  MoveC 574 to (267.87, -55.04, -8.35) mm, rotated rx -180 ry 0 rz 0 deg; joints [19.614, -51.076, 148.071, 19.71, -95.718, 2.626] to (268.06, -55.49, -8.35) mm, rotated rx -180 ry 0 rz 0 deg; joints [19.592, -51.078, 148.094, 19.688, -95.739, 2.631]
  MoveL 575 to (268.06, -80.89, -8.35) mm, rotated rx -180 ry 0 rz 0 deg; joints [18.101, -51.105, 148.664, 18.209, -96.314, 2.629]
  MoveL 576 to (217.26, -80.89, -8.35) mm, rotated rx -180 ry 0 rz 0 deg; joints [17.167, -50.698, 145.241, 17.193, -93.471, 1.614]
  MoveL 577 to (217.26, -30.09, -8.35) mm, rotated rx 180 ry 0 rz 0 deg; joints [19.994, -50.561, 144.093, 20.006, -92.45, 1.48]
  MoveL 578 to (268.06, -30.09, -8.35) mm, rotated rx 180 ry 0 rz 0 deg; joints [21.056, -51.039, 147.478, 21.138, -95.138, 2.59]
  MoveL 579 to (268.06, -55.49, -8.35) mm, rotated rx -180 ry 0 rz 0 deg; joints [19.592, -51.078, 148.094, 19.688, -95.739, 2.631]
  MoveC 580 to (267.87, -55.94, -8.35) mm, rotated rx 180 ry 0 rz 0 deg; joints [19.562, -51.077, 148.092, 19.658, -95.739, 2.627] to (267.42, -56.12, -8.35) mm, rotated rx -180 ry 0 rz 0 deg; joints [19.542, -51.074, 148.066, 19.637, -95.719, 2.617]
  MoveL 581 to (266.79, -56.12, -8.35) mm, rotated rx 180 ry 0 rz 0 deg; joints [19.529, -51.07, 148.024, 19.623, -95.684, 2.603]
  MoveC 582 to (266.34, -56.12, -8.16) mm, rotated rx -180 ry 0 rz 0 deg; joints [19.519, -51.086, 147.998, 19.612, -95.645, 2.588] to (266.15, -56.12, -7.72) mm, rotated rx -180 ry 0 rz 0 deg; joints [19.515, -51.13, 147.995, 19.606, -95.6, 2.571]
  Set speed (500.0 mm/s)
  MoveL 583 to (266.15, -56.12, 6) mm, rotated rx 180 ry 0 rz 0 deg; joints [19.507, -52.51, 148.253, 19.565, -94.544, 2.193]
  MoveL 584 to (139.15, -54.85, 6) mm, rotated rx 180 ry 0 rz 0 deg; joints [17.26, -50.798, 139.522, 17.265, -87.911, -0.107]
  Set speed (25.4 mm/s)
  MoveL 585 to (139.15, -54.85, -3.54) mm, rotated rx -180 ry 0 rz 0 deg; joints [17.264, -49.983, 139.368, 17.264, -88.543, 0.09]
  MoveC 586 to (139.34, -54.85, -3.99) mm, rotated rx 180 ry 0 rz 0 deg; joints [17.268, -49.948, 139.374, 17.267, -88.582, 0.102] to (139.79, -54.85, -4.17) mm, rotated rx -180 ry 0 rz 0 deg; joints [17.275, -49.94, 139.402, 17.274, -88.617, 0.113]
  Set speed (50.8 mm/s)
  MoveL 587 to (140.42, -54.85, -4.18) mm, rotated rx 180 ry 0 rz 0 deg; joints [17.285, -49.95, 139.447, 17.284, -88.65, 0.123]
  MoveC 588 to (140.87, -55.04, -4.18) mm, rotated rx -180 ry 0 rz 0 deg; joints [17.283, -49.958, 139.482, 17.281, -88.676, 0.131] to (141.06, -55.49, -4.17) mm, rotated rx -180 ry 0 rz 0 deg; joints [17.262, -49.963, 139.505, 17.261, -88.693, 0.136]
  MoveL 589 to (141.06, -80.89, -4.17) mm, rotated rx 180 ry 0 rz 0 deg; joints [15.927, -50.066, 140.034, 15.923, -89.099, 0.263]
  MoveL 590 to (90.26, -80.89, -4.18) mm, rotated rx -180 ry 0 rz 0 deg; joints [15.195, -49.17, 136.413, 15.218, -86.47, -0.451]
  MoveL 591 to (90.26, -30.09, -4.18) mm, rotated rx -180 ry 0 rz 0 deg; joints [17.739, -48.917, 135.342, 17.784, -85.727, -0.819]
  MoveL 592 to (141.06, -30.09, -4.17) mm, rotated rx -180 ry 0 rz 0 deg; joints [18.578, -49.847, 138.934, 18.581, -88.265, -0.019]
  MoveL 593 to (141.06, -55.49, -4.18) mm, rotated rx -180 ry 0 rz 0 deg; joints [17.262, -49.963, 139.505, 17.261, -88.693, 0.136]
  MoveC 594 to (140.87, -55.94, -4.18) mm, rotated rx 180 ry 0 rz 0 deg; joints [17.236, -49.962, 139.502, 17.234, -88.691, 0.136] to (140.42, -56.12, -4.17) mm, rotated rx -180 ry 0 rz 0 deg; joints [17.219, -49.956, 139.474, 17.218, -88.671, 0.13]
  MoveL 595 to (139.79, -56.12, -4.18) mm, rotated rx 180 ry 0 rz 0 deg; joints [17.209, -49.945, 139.43, 17.208, -88.638, 0.12]
  MoveC 596 to (139.34, -56.12, -3.99) mm, rotated rx -180 ry 0 rz 0 deg; joints [17.201, -49.954, 139.401, 17.2, -88.603, 0.109] to (139.15, -56.12, -3.54) mm, rotated rx -180 ry 0 rz 0 deg; joints [17.198, -49.989, 139.396, 17.198, -88.564, 0.097]
  Set speed (500.0 mm/s)
  MoveL 597 to (139.15, -56.12, 5) mm, rotated rx -180 ry 0 rz 0 deg; joints [17.194, -50.719, 139.534, 17.199, -87.998, -0.078]
  MoveL 598 to (139.15, -54.85, 5) mm, rotated rx -180 ry 0 rz 0 deg; joints [17.26, -50.713, 139.506, 17.265, -87.978, -0.086]
  Set speed (25.4 mm/s)
  MoveL 599 to (139.15, -54.85, 1.82) mm, rotated rx -180 ry 0 rz 0 deg; joints [17.262, -50.442, 139.456, 17.264, -88.189, -0.02]
  MoveL 600 to (139.15, -54.85, -7.72) mm, rotated rx -180 ry 0 rz 0 deg; joints [17.266, -49.627, 139.298, 17.264, -88.817, 0.175]
  MoveC 601 to (139.34, -54.85, -8.16) mm, rotated rx 180 ry 0 rz 0 deg; joints [17.27, -49.591, 139.304, 17.267, -88.856, 0.187] to (139.79, -54.85, -8.35) mm, rotated rx -180 ry 0 rz 0 deg; joints [17.277, -49.583, 139.332, 17.274, -88.891, 0.198]
  Set speed (50.8 mm/s)
  MoveL 602 to (140.42, -54.85, -8.35) mm, rotated rx 180 ry 0 rz 0 deg; joints [17.287, -49.593, 139.377, 17.284, -88.924, 0.208]
  MoveC 603 to (140.87, -55.04, -8.35) mm, rotated rx 180 ry 0 rz 0 deg; joints [17.285, -49.601, 139.412, 17.282, -88.95, 0.216] to (141.06, -55.49, -8.35) mm, rotated rx -180 ry 0 rz 0 deg; joints [17.264, -49.606, 139.435, 17.261, -88.967, 0.222]
  MoveL 604 to (141.06, -80.89, -8.35) mm, rotated rx -180 ry 0 rz 0 deg; joints [15.929, -49.706, 139.963, 15.924, -89.378, 0.343]
  MoveL 605 to (90.26, -80.89, -8.35) mm, rotated rx 180 ry 0 rz 0 deg; joints [15.197, -48.831, 136.346, 15.216, -86.732, -0.38]
  MoveL 606 to (90.26, -30.09, -8.35) mm, rotated rx 180 ry 0 rz 0 deg; joints [17.741, -48.582, 135.276, 17.78, -85.981, -0.737]
  MoveL 607 to (141.06, -30.09, -8.35) mm, rotated rx -180 ry 0 rz 0 deg; joints [18.58, -49.493, 138.864, 18.58, -88.534, 0.072]
  MoveL 608 to (141.06, -55.49, -8.35) mm, rotated rx -180 ry 0 rz 0 deg; joints [17.264, -49.606, 139.435, 17.261, -88.967, 0.222]
  MoveC 609 to (140.87, -55.94, -8.35) mm, rotated rx -180 ry 0 rz 0 deg; joints [17.238, -49.605, 139.431, 17.235, -88.965, 0.221] to (140.42, -56.12, -8.35) mm, rotated rx 180 ry 0 rz 0 deg; joints [17.221, -49.598, 139.404, 17.218, -88.945, 0.215]
  MoveL 610 to (139.79, -56.12, -8.35) mm, rotated rx 180 ry 0 rz 0 deg; joints [17.211, -49.588, 139.359, 17.208, -88.912, 0.205]
  MoveC 611 to (139.34, -56.12, -8.16) mm, rotated rx -180 ry 0 rz 0 deg; joints [17.203, -49.597, 139.331, 17.201, -88.877, 0.194] to (139.15, -56.12, -7.72) mm, rotated rx 180 ry 0 rz 0 deg; joints [17.2, -49.632, 139.326, 17.198, -88.838, 0.182]
  Set speed (500.0 mm/s)
  MoveL 612 to (139.15, -56.12, 6) mm, rotated rx -180 ry 0 rz 0 deg; joints [17.193, -50.804, 139.549, 17.199, -87.931, -0.099]
  MoveL 613 to (139.15, -235.88, 6) mm, rotated rx -180 ry 0 rz 0 deg; joints [7.42, -51.334, 142.34, 7.415, -90.128, 0.402]
  Set speed (25.4 mm/s)
  MoveL 614 to (139.15, -235.88, -3.54) mm, rotated rx -180 ry 0 rz 0 deg; joints [7.424, -50.477, 142.179, 7.42, -90.818, 0.492]
  MoveC 615 to (139.34, -235.88, -3.99) mm, rotated rx -180 ry 0 rz 0 deg; joints [7.425, -50.44, 142.185, 7.421, -90.861, 0.498] to (139.79, -235.88, -4.17) mm, rotated rx -180 ry 0 rz 0 deg; joints [7.429, -50.43, 142.214, 7.425, -90.9, 0.503]
  Set speed (50.8 mm/s)
  MoveL 616 to (140.42, -235.88, -4.18) mm, rotated rx -180 ry 0 rz 0 deg; joints [7.433, -50.439, 142.259, 7.429, -90.936, 0.508]
  MoveC 617 to (140.87, -236.07, -4.17) mm, rotated rx 180 ry 0 rz 0 deg; joints [7.426, -50.445, 142.293, 7.422, -90.963, 0.511] to (141.06, -236.52, -4.17) mm, rotated rx -180 ry 0 rz 0 deg; joints [7.402, -50.448, 142.311, 7.398, -90.977, 0.512]
  MoveL 618 to (141.06, -261.92, -4.18) mm, rotated rx 180 ry 0 rz 0 deg; joints [5.968, -50.475, 142.522, 5.965, -91.166, 0.485]
  MoveL 619 to (90.26, -261.92, -4.18) mm, rotated rx -180 ry 0 rz 0 deg; joints [5.682, -49.673, 138.831, 5.68, -88.293, 0.189]
  MoveL 620 to (90.26, -211.12, -4.18) mm, rotated rx 180 ry 0 rz 0 deg; joints [8.407, -49.59, 138.377, 8.407, -87.931, 0.095]
  MoveL 621 to (141.06, -211.12, -4.18) mm, rotated rx -180 ry 0 rz 0 deg; joints [8.827, -50.412, 142.054, 8.822, -90.753, 0.524]
  MoveL 622 to (141.06, -236.52, -4.17) mm, rotated rx -180 ry 0 rz 0 deg; joints [7.402, -50.448, 142.311, 7.398, -90.977, 0.512]
  MoveC 623 to (140.87, -236.97, -4.18) mm, rotated rx -180 ry 0 rz 0 deg; joints [7.376, -50.446, 142.302, 7.372, -90.97, 0.51] to (140.42, -237.16, -4.17) mm, rotated rx 180 ry 0 rz 0 deg; joints [7.362, -50.44, 142.271, 7.358, -90.946, 0.507]
  MoveL 624 to (139.79, -237.15, -4.18) mm, rotated rx -180 ry 0 rz 0 deg; joints [7.357, -50.431, 142.225, 7.353, -90.91, 0.502]
  MoveC 625 to (139.34, -237.15, -3.99) mm, rotated rx -180 ry 0 rz 0 deg; joints [7.354, -50.441, 142.196, 7.35, -90.871, 0.497] to (139.15, -237.15, -3.54) mm, rotated rx -180 ry 0 rz 0 deg; joints [7.352, -50.479, 142.191, 7.348, -90.828, 0.491]
  Set speed (500.0 mm/s)
  MoveL 626 to (139.15, -237.16, 5) mm, rotated rx -180 ry 0 rz 0 deg; joints [7.349, -51.246, 142.335, 7.344, -90.211, 0.412]
  MoveL 627 to (139.15, -235.89, 5) mm, rotated rx -180 ry 0 rz 0 deg; joints [7.421, -51.244, 142.323, 7.416, -90.201, 0.412]
  Set speed (25.4 mm/s)
  MoveL 628 to (139.15, -235.88, 1.83) mm, rotated rx -180 ry 0 rz 0 deg; joints [7.422, -50.959, 142.271, 7.417, -90.431, 0.442]
  MoveL 629 to (139.15, -235.89, -7.72) mm, rotated rx 180 ry 0 rz 0 deg; joints [7.425, -50.103, 142.106, 7.422, -91.117, 0.531]
  MoveC 630 to (139.34, -235.89, -8.16) mm, rotated rx -180 ry 0 rz 0 deg; joints [7.427, -50.065, 142.111, 7.423, -91.16, 0.537] to (139.79, -235.88, -8.35) mm, rotated rx -180 ry 0 rz 0 deg; joints [7.43, -50.055, 142.14, 7.427, -91.199, 0.542]
  Set speed (50.8 mm/s)
  MoveL 631 to (140.42, -235.88, -8.35) mm, rotated rx 180 ry 0 rz 0 deg; joints [7.435, -50.063, 142.186, 7.432, -91.235, 0.547]
  MoveC 632 to (140.87, -236.07, -8.35) mm, rotated rx 180 ry 0 rz 0 deg; joints [7.428, -50.07, 142.22, 7.425, -91.262, 0.55] to (141.06, -236.52, -8.35) mm, rotated rx -180 ry 0 rz 0 deg; joints [7.404, -50.073, 142.237, 7.401, -91.277, 0.551]
  MoveL 633 to (141.06, -261.92, -8.35) mm, rotated rx -180 ry 0 rz 0 deg; joints [5.97, -50.098, 142.448, 5.967, -91.467, 0.517]
  MoveL 634 to (90.26, -261.92, -8.35) mm, rotated rx -180 ry 0 rz 0 deg; joints [5.684, -49.319, 138.761, 5.681, -88.576, 0.217]
  MoveL 635 to (90.26, -211.12, -8.35) mm, rotated rx 180 ry 0 rz 0 deg; joints [8.409, -49.239, 138.308, 8.408, -88.209, 0.136]
  MoveL 636 to (141.06, -211.12, -8.35) mm, rotated rx -180 ry 0 rz 0 deg; joints [8.829, -50.038, 141.981, 8.825, -91.05, 0.57]
  MoveL 637 to (141.06, -236.52, -8.35) mm, rotated rx -180 ry 0 rz 0 deg; joints [7.404, -50.073, 142.237, 7.401, -91.277, 0.551]
  MoveC 638 to (140.87, -236.97, -8.35) mm, rotated rx -180 ry 0 rz 0 deg; joints [7.377, -50.071, 142.228, 7.374, -91.27, 0.549] to (140.42, -237.16, -8.35) mm, rotated rx 180 ry 0 rz 0 deg; joints [7.363, -50.065, 142.197, 7.36, -91.246, 0.546]
  MoveL 639 to (139.79, -237.15, -8.35) mm, rotated rx -180 ry 0 rz 0 deg; joints [7.359, -50.056, 142.152, 7.356, -91.209, 0.541]
  MoveC 640 to (139.34, -237.15, -8.16) mm, rotated rx -180 ry 0 rz 0 deg; joints [7.356, -50.067, 142.123, 7.352, -91.17, 0.535] to (139.15, -237.16, -7.72) mm, rotated rx -180 ry 0 rz 0 deg; joints [7.354, -50.104, 142.118, 7.35, -91.127, 0.53]
  Set speed (500.0 mm/s)
  MoveL 641 to (139.15, -237.15, 6) mm, rotated rx -180 ry 0 rz 0 deg; joints [7.349, -51.336, 142.351, 7.344, -90.138, 0.402]
  MoveL 642 to (266.15, -235.88, 6) mm, rotated rx 180 ry 0 rz 0 deg; joints [8.48, -52.646, 151.287, 8.552, -97.677, 1.553]
  Set speed (25.4 mm/s)
  MoveL 643 to (266.15, -235.88, -3.54) mm, rotated rx -180 ry 0 rz 0 deg; joints [8.485, -51.621, 151.098, 8.574, -98.503, 1.679]
  MoveC 644 to (266.34, -235.88, -3.99) mm, rotated rx -180 ry 0 rz 0 deg; joints [8.487, -51.573, 151.102, 8.578, -98.554, 1.687] to (266.79, -235.89, -4.17) mm, rotated rx 180 ry 0 rz 0 deg; joints [8.491, -51.555, 151.128, 8.583, -98.599, 1.695]
  Set speed (50.8 mm/s)
  MoveL 645 to (267.42, -235.88, -4.18) mm, rotated rx -180 ry 0 rz 0 deg; joints [8.497, -51.556, 151.172, 8.59, -98.64, 1.702]
  MoveC 646 to (267.87, -236.07, -4.18) mm, rotated rx -180 ry 0 rz 0 deg; joints [8.489, -51.557, 151.205, 8.583, -98.672, 1.706] to (268.06, -236.52, -4.17) mm, rotated rx 180 ry 0 rz 0 deg; joints [8.462, -51.557, 151.222, 8.556, -98.689, 1.704]
  MoveL 647 to (268.06, -261.92, -4.17) mm, rotated rx -180 ry 0 rz 0 deg; joints [6.827, -51.546, 151.452, 6.907, -98.966, 1.458]
  MoveL 648 to (217.26, -261.92, -4.18) mm, rotated rx -180 ry 0 rz 0 deg; joints [6.456, -51.304, 147.93, 6.483, -95.714, 1.019]
  MoveL 649 to (217.26, -211.12, -4.17) mm, rotated rx -180 ry 0 rz 0 deg; joints [9.541, -51.283, 147.438, 9.575, -95.2, 1.294]
  MoveL 650 to (268.06, -211.12, -4.17) mm, rotated rx 180 ry 0 rz 0 deg; joints [10.084, -51.566, 150.942, 10.188, -98.36, 1.924]
  MoveL 651 to (268.06, -236.52, -4.17) mm, rotated rx 180 ry 0 rz 0 deg; joints [8.462, -51.557, 151.222, 8.556, -98.689, 1.704]
  MoveC 652 to (267.87, -236.97, -4.17) mm, rotated rx -180 ry 0 rz 0 deg; joints [8.432, -51.557, 151.214, 8.525, -98.682, 1.697] to (267.42, -237.15, -4.17) mm, rotated rx -180 ry 0 rz 0 deg; joints [8.416, -51.556, 151.185, 8.508, -98.655, 1.691]
  MoveL 653 to (266.79, -237.16, -4.17) mm, rotated rx 180 ry 0 rz 0 deg; joints [8.41, -51.554, 151.141, 8.501, -98.614, 1.683]
  MoveC 654 to (266.34, -237.15, -3.99) mm, rotated rx -180 ry 0 rz 0 deg; joints [8.405, -51.573, 151.114, 8.496, -98.569, 1.676] to (266.15, -237.15, -3.54) mm, rotated rx -180 ry 0 rz 0 deg; joints [8.403, -51.621, 151.111, 8.493, -98.518, 1.668]
  Set speed (500.0 mm/s)
  MoveL 655 to (266.15, -237.15, 5) mm, rotated rx -180 ry 0 rz 0 deg; joints [8.399, -52.538, 151.281, 8.473, -97.779, 1.556]
  MoveL 656 to (266.15, -235.88, 5) mm, rotated rx -180 ry 0 rz 0 deg; joints [8.481, -52.538, 151.268, 8.555, -97.764, 1.566]
  Set speed (25.4 mm/s)
  MoveL 657 to (266.15, -235.88, 1.82) mm, rotated rx -180 ry 0 rz 0 deg; joints [8.482, -52.197, 151.206, 8.562, -98.04, 1.608]
  MoveL 658 to (266.15, -235.88, -7.72) mm, rotated rx 180 ry 0 rz 0 deg; joints [8.486, -51.174, 151.012, 8.585, -98.86, 1.734]
  MoveC 659 to (266.34, -235.89, -8.16) mm, rotated rx 180 ry 0 rz 0 deg; joints [8.488, -51.126, 151.015, 8.588, -98.91, 1.742] to (266.79, -235.89, -8.35) mm, rotated rx -180 ry 0 rz 0 deg; joints [8.493, -51.107, 151.042, 8.593, -98.956, 1.75]
  Set speed (50.8 mm/s)
  MoveL 660 to (267.42, -235.88, -8.35) mm, rotated rx -180 ry 0 rz 0 deg; joints [8.499, -51.108, 151.085, 8.6, -98.997, 1.757]
  MoveC 661 to (267.87, -236.07, -8.35) mm, rotated rx -180 ry 0 rz 0 deg; joints [8.491, -51.109, 151.118, 8.593, -99.029, 1.761] to (268.06, -236.52, -8.35) mm, rotated rx -180 ry 0 rz 0 deg; joints [8.464, -51.109, 151.135, 8.566, -99.047, 1.759]
  MoveL 662 to (268.06, -261.92, -8.35) mm, rotated rx -180 ry 0 rz 0 deg; joints [6.829, -51.095, 151.365, 6.916, -99.327, 1.503]
  MoveL 663 to (217.26, -261.92, -8.35) mm, rotated rx 180 ry 0 rz 0 deg; joints [6.457, -50.886, 147.848, 6.489, -96.049, 1.057]
  MoveL 664 to (217.26, -211.12, -8.35) mm, rotated rx -180 ry 0 rz 0 deg; joints [9.543, -50.869, 147.358, 9.582, -95.529, 1.35]
  MoveL 665 to (268.06, -211.12, -8.35) mm, rotated rx -180 ry 0 rz 0 deg; joints [10.086, -51.121, 150.856, 10.2, -98.714, 1.988]
  MoveL 666 to (268.06, -236.52, -8.35) mm, rotated rx -180 ry 0 rz 0 deg; joints [8.464, -51.109, 151.135, 8.566, -99.047, 1.759]
  MoveC 667 to (267.87, -236.97, -8.35) mm, rotated rx 180 ry 0 rz 0 deg; joints [8.434, -51.108, 151.127, 8.535, -99.04, 1.752] to (267.42, -237.16, -8.35) mm, rotated rx -180 ry 0 rz 0 deg; joints [8.417, -51.107, 151.098, 8.518, -99.013, 1.745]
  MoveL 668 to (266.79, -237.16, -8.35) mm, rotated rx 180 ry 0 rz 0 deg; joints [8.411, -51.106, 151.054, 8.511, -98.971, 1.738]
  MoveC 669 to (266.34, -237.16, -8.16) mm, rotated rx -180 ry 0 rz 0 deg; joints [8.407, -51.125, 151.028, 8.506, -98.926, 1.73] to (266.15, -237.16, -7.72) mm, rotated rx -180 ry 0 rz 0 deg; joints [8.405, -51.173, 151.024, 8.503, -98.875, 1.722]
  Set speed (500.0 mm/s)
  MoveL 670 to (266.15, -237.15, 6) mm, rotated rx 180 ry 0 rz 0 deg; joints [8.399, -52.646, 151.3, 8.471, -97.692, 1.543]
  MoveL 671 to (393.15, -235.88, 6) mm, rotated rx -180 ry 0 rz -30 deg; joints [-2.476, -52.361, 157.47, -33.311, -102.092, -7.56]
  Set speed (25.4 mm/s)
  MoveL 672 to (393.15, -235.88, -3.54) mm, rotated rx -180 ry 0 rz -30 deg; joints [-2.473, -51.174, 157.249, -33.426, -102.899, -8.104]
  MoveC 673 to (393.34, -235.88, -3.99) mm, rotated rx -180 ry 0 rz -30 deg; joints [-2.474, -51.116, 157.251, -33.434, -102.949, -8.138] to (393.79, -235.88, -4.17) mm, rotated rx 180 ry 0 rz -30 deg; joints [-2.475, -51.088, 157.277, -33.442, -102.994, -8.168]
  Set speed (50.8 mm/s)
  MoveL 674 to (394.42, -235.88, -4.17) mm, rotated rx -180 ry 0 rz -30 deg; joints [-2.477, -51.08, 157.319, -33.45, -103.035, -8.197]
  MoveC 675 to (394.87, -236.07, -4.17) mm, rotated rx -180 ry 0 rz -30 deg; joints [-2.492, -51.075, 157.349, -33.47, -103.061, -8.22] to (395.06, -236.52, -4.18) mm, rotated rx 180 ry 0 rz -30 deg; joints [-2.525, -51.073, 157.36, -33.505, -103.067, -8.236]
  MoveL 676 to (395.06, -261.92, -4.17) mm, rotated rx 180 ry 0 rz -30 deg; joints [-4.354, -51.079, 157.255, -35.344, -102.688, -8.604]
  MoveL 677 to (344.26, -261.92, -4.17) mm, rotated rx -180 ry 0 rz 0 deg; joints [7.472, -51.287, 156.609, 7.707, -104.32, 2.303]
  MoveL 678 to (344.26, -211.12, -4.18) mm, rotated rx 180 ry 0 rz 0 deg; joints [11.024, -51.402, 156.068, 11.337, -103.521, 3.125]
  MoveL 679 to (395.06, -211.12, -4.17) mm, rotated rx 180 ry 0 rz -30 deg; joints [-0.69, -51.078, 157.41, -31.648, -103.383, -7.814]
  MoveL 680 to (395.06, -236.52, -4.18) mm, rotated rx 180 ry 0 rz -30 deg; joints [-2.525, -51.073, 157.36, -33.505, -103.067, -8.236]
  MoveC 681 to (394.87, -236.97, -4.18) mm, rotated rx -180 ry 0 rz -30 deg; joints [-2.556, -51.075, 157.346, -33.535, -103.049, -8.234] to (394.42, -237.16, -4.18) mm, rotated rx 180 ry 0 rz -30 deg; joints [-2.568, -51.08, 157.315, -33.543, -103.017, -8.217]
  MoveL 682 to (393.79, -237.16, -4.18) mm, rotated rx 180 ry 0 rz -30 deg; joints [-2.566, -51.088, 157.273, -33.534, -102.976, -8.188]
  MoveC 683 to (393.34, -237.16, -3.99) mm, rotated rx 180 ry 0 rz -30 deg; joints [-2.565, -51.116, 157.247, -33.526, -102.932, -8.157] to (393.15, -237.15, -3.54) mm, rotated rx -180 ry 0 rz -30 deg; joints [-2.564, -51.174, 157.246, -33.518, -102.882, -8.123]
  Set speed (500.0 mm/s)
  MoveL 684 to (393.15, -237.15, 5) mm, rotated rx -180 ry 0 rz -30 deg; joints [-2.567, -52.236, 157.444, -33.415, -102.161, -7.636]
  MoveL 685 to (393.15, -235.88, 5) mm, rotated rx 180 ry 0 rz -30 deg; joints [-2.476, -52.236, 157.448, -33.323, -102.177, -7.617]
  Set speed (25.4 mm/s)
  MoveL 686 to (393.15, -235.88, 1.83) mm, rotated rx 180 ry 0 rz -30 deg; joints [-2.475, -51.84, 157.375, -33.36, -102.447, -7.799]
  MoveL 687 to (393.15, -235.89, -7.72) mm, rotated rx -180 ry 0 rz -30 deg; joints [-2.472, -50.657, 157.149, -33.478, -103.247, -8.339]
  MoveC 688 to (393.34, -235.89, -8.16) mm, rotated rx 180 ry 0 rz -30 deg; joints [-2.472, -50.599, 157.15, -33.486, -103.296, -8.373] to (393.79, -235.89, -8.35) mm, rotated rx -180 ry 0 rz -30 deg; joints [-2.474, -50.571, 157.176, -33.494, -103.341, -8.404]
  Set speed (50.8 mm/s)
  MoveL 689 to (394.42, -235.88, -8.35) mm, rotated rx -180 ry 0 rz -30 deg; joints [-2.476, -50.563, 157.218, -33.503, -103.382, -8.433]
  MoveC 690 to (394.87, -236.07, -8.35) mm, rotated rx -180 ry 0 rz -30 deg; joints [-2.49, -50.557, 157.247, -33.523, -103.409, -8.456] to (395.06, -236.52, -8.35) mm, rotated rx -180 ry 0 rz -30 deg; joints [-2.523, -50.555, 157.258, -33.558, -103.415, -8.472]
  MoveL 691 to (395.06, -261.92, -8.35) mm, rotated rx -180 ry 0 rz -30 deg; joints [-4.353, -50.562, 157.154, -35.398, -103.027, -8.851]
  MoveL 692 to (344.26, -261.92, -8.35) mm, rotated rx -180 ry 0 rz 0 deg; joints [7.474, -50.779, 156.51, 7.724, -104.726, 2.361]
  MoveL 693 to (344.26, -211.12, -8.35) mm, rotated rx -180 ry 0 rz 0 deg; joints [11.026, -50.9, 155.971, 11.358, -103.917, 3.208]
  MoveL 694 to (395.06, -211.12, -8.35) mm, rotated rx 180 ry 0 rz -30 deg; joints [-0.689, -50.559, 157.309, -31.699, -103.738, -8.04]
  MoveL 695 to (395.06, -236.52, -8.35) mm, rotated rx 180 ry 0 rz -30 deg; joints [-2.523, -50.555, 157.258, -33.558, -103.415, -8.472]
  MoveC 696 to (394.87, -236.97, -8.35) mm, rotated rx -180 ry 0 rz -30 deg; joints [-2.555, -50.557, 157.245, -33.588, -103.397, -8.471] to (394.42, -237.16, -8.35) mm, rotated rx -180 ry 0 rz -30 deg; joints [-2.567, -50.563, 157.214, -33.595, -103.365, -8.453]
  MoveL 697 to (393.79, -237.15, -8.35) mm, rotated rx -180 ry 0 rz -30 deg; joints [-2.565, -50.571, 157.172, -33.587, -103.323, -8.424]
  MoveC 698 to (393.34, -237.15, -8.16) mm, rotated rx -180 ry 0 rz -30 deg; joints [-2.564, -50.599, 157.147, -33.578, -103.279, -8.393] to (393.15, -237.16, -7.72) mm, rotated rx -180 ry 0 rz -30 deg; joints [-2.563, -50.657, 157.145, -33.57, -103.229, -8.359]
  Set speed (500.0 mm/s)
  MoveL 699 to (393.15, -237.16, 6) mm, rotated rx 180 ry 0 rz -30 deg; joints [-2.567, -52.361, 157.466, -33.403, -102.075, -7.578]
  MoveL 700 to (393.15, -422.22, 6) mm, rotated rx 180 ry 0 rz -30 deg; joints [-15.522, -52.504, 155.473, -46.167, -98.438, -8.647]
  Set speed (25.4 mm/s)
  MoveL 701 to (393.15, -422.22, -3.54) mm, rotated rx 180 ry 0 rz -30 deg; joints [-15.522, -51.374, 155.264, -46.269, -99.074, -9.319]
  MoveC 702 to (393.34, -422.22, -3.99) mm, rotated rx -180 ry 0 rz -30 deg; joints [-15.526, -51.32, 155.266, -46.279, -99.112, -9.361] to (393.79, -422.22, -4.17) mm, rotated rx 180 ry 0 rz -30 deg; joints [-15.534, -51.295, 155.291, -46.293, -99.145, -9.399]
  Set speed (50.8 mm/s)
  MoveL 703 to (394.42, -422.22, -4.18) mm, rotated rx -180 ry 0 rz -30 deg; joints [-15.546, -51.291, 155.332, -46.31, -99.174, -9.434]
  MoveC 704 to (394.87, -422.41, -4.17) mm, rotated rx -180 ry 0 rz -30 deg; joints [-15.567, -51.289, 155.358, -46.334, -99.19, -9.458] to (395.06, -422.86, -4.18) mm, rotated rx -180 ry 0 rz -30 deg; joints [-15.6, -51.288, 155.362, -46.368, -99.188, -9.467]
  MoveL 705 to (395.06, -448.26, -4.17) mm, rotated rx -180 ry 0 rz -30 deg; joints [-17.289, -51.33, 154.874, -47.991, -98.532, -9.352]
  MoveL 706 to (344.26, -448.26, -4.18) mm, rotated rx -180 ry 0 rz 0 deg; joints [-5.845, -51.148, 156.765, -6.046, -104.665, -1.353]
  MoveL 707 to (344.26, -397.46, -4.17) mm, rotated rx -180 ry 0 rz 0 deg; joints [-2.217, -51.134, 157.009, -2.299, -104.994, -0.356]
  MoveL 708 to (395.06, -397.46, -4.18) mm, rotated rx 180 ry 0 rz -30 deg; joints [-13.883, -51.245, 155.799, -44.712, -99.827, -9.513]
  MoveL 709 to (395.06, -422.86, -4.18) mm, rotated rx -180 ry 0 rz -30 deg; joints [-15.6, -51.288, 155.362, -46.368, -99.188, -9.467]
  MoveC 710 to (394.87, -423.31, -4.18) mm, rotated rx -180 ry 0 rz -30 deg; joints [-15.627, -51.29, 155.342, -46.392, -99.168, -9.455] to (394.42, -423.49, -4.17) mm, rotated rx -180 ry 0 rz -30 deg; joints [-15.631, -51.293, 155.309, -46.392, -99.142, -9.43]
  MoveL 711 to (393.79, -423.49, -4.17) mm, rotated rx 180 ry 0 rz -30 deg; joints [-15.619, -51.297, 155.268, -46.375, -99.113, -9.395]
  MoveC 712 to (393.34, -423.49, -3.99) mm, rotated rx -180 ry 0 rz -30 deg; joints [-15.611, -51.322, 155.243, -46.361, -99.08, -9.357] to (393.15, -423.49, -3.54) mm, rotated rx 180 ry 0 rz -30 deg; joints [-15.607, -51.376, 155.241, -46.351, -99.042, -9.315]
  Set speed (500.0 mm/s)
  MoveL 713 to (393.15, -423.49, 5) mm, rotated rx 180 ry 0 rz -30 deg; joints [-15.607, -52.386, 155.429, -46.259, -98.474, -8.714]
  MoveL 714 to (393.15, -422.22, 5) mm, rotated rx -180 ry 0 rz -30 deg; joints [-15.522, -52.385, 155.452, -46.177, -98.505, -8.718]
  Set speed (25.4 mm/s)
  MoveL 715 to (393.15, -422.22, 1.83) mm, rotated rx 180 ry 0 rz -30 deg; joints [-15.522, -52.008, 155.383, -46.211, -98.718, -8.943]
  MoveL 716 to (393.15, -422.22, -7.72) mm, rotated rx -180 ry 0 rz -30 deg; joints [-15.522, -50.882, 155.168, -46.315, -99.348, -9.61]
  MoveC 717 to (393.34, -422.22, -8.16) mm, rotated rx 180 ry 0 rz -30 deg; joints [-15.525, -50.828, 155.17, -46.325, -99.386, -9.651] to (393.79, -422.22, -8.35) mm, rotated rx -180 ry 0 rz -30 deg; joints [-15.534, -50.803, 155.195, -46.34, -99.419, -9.689]
  Set speed (50.8 mm/s)
  MoveL 718 to (394.42, -422.22, -8.35) mm, rotated rx -180 ry 0 rz -30 deg; joints [-15.546, -50.798, 155.236, -46.357, -99.449, -9.725]
  MoveC 719 to (394.87, -422.41, -8.35) mm, rotated rx -180 ry 0 rz -30 deg; joints [-15.566, -50.795, 155.262, -46.381, -99.465, -9.749] to (395.06, -422.86, -8.35) mm, rotated rx -180 ry 0 rz -30 deg; joints [-15.6, -50.795, 155.266, -46.415, -99.462, -9.758]
  MoveL 720 to (395.06, -448.26, -8.35) mm, rotated rx -180 ry 0 rz -30 deg; joints [-17.289, -50.842, 154.78, -48.035, -98.795, -9.647]
  MoveL 721 to (344.26, -448.26, -8.35) mm, rotated rx -180 ry 0 rz 0 deg; joints [-5.844, -50.638, 156.666, -6.057, -105.073, -1.397]
  MoveL 722 to (344.26, -397.46, -8.35) mm, rotated rx -180 ry 0 rz 0 deg; joints [-2.216, -50.62, 156.909, -2.302, -105.407, -0.373]
  MoveL 723 to (395.06, -397.46, -8.35) mm, rotated rx -180 ry 0 rz -30 deg; joints [-13.883, -50.746, 155.702, -44.761, -100.112, -9.8]
  MoveL 724 to (395.06, -422.86, -8.35) mm, rotated rx -180 ry 0 rz -30 deg; joints [-15.6, -50.795, 155.266, -46.415, -99.462, -9.758]
  MoveC 725 to (394.87, -423.31, -8.35) mm, rotated rx -180 ry 0 rz -30 deg; joints [-15.627, -50.797, 155.246, -46.439, -99.441, -9.747] to (394.42, -423.49, -8.35) mm, rotated rx 180 ry 0 rz -30 deg; joints [-15.631, -50.801, 155.213, -46.439, -99.416, -9.721]
  MoveL 726 to (393.79, -423.49, -8.35) mm, rotated rx -180 ry 0 rz -30 deg; joints [-15.619, -50.805, 155.172, -46.421, -99.386, -9.685]
  MoveC 727 to (393.34, -423.49, -8.16) mm, rotated rx -180 ry 0 rz -30 deg; joints [-15.61, -50.83, 155.147, -46.407, -99.354, -9.647] to (393.15, -423.49, -7.72) mm, rotated rx -180 ry 0 rz -30 deg; joints [-15.607, -50.884, 155.145, -46.397, -99.316, -9.606]
  Set speed (500.0 mm/s)
  MoveL 728 to (393.15, -423.49, 6) mm, rotated rx -180 ry 0 rz -30 deg; joints [-15.607, -52.505, 155.45, -46.249, -98.407, -8.643]
  MoveL 729 to (266.15, -422.22, 6) mm, rotated rx -180 ry 0 rz 0 deg; joints [-3.637, -52.566, 151.817, -3.68, -98.363, -0.319]
  Set speed (25.4 mm/s)
  MoveL 730 to (266.15, -422.22, -3.54) mm, rotated rx 180 ry 0 rz 0 deg; joints [-3.635, -51.529, 151.625, -3.686, -99.206, -0.373]
  MoveC 731 to (266.34, -422.22, -3.99) mm, rotated rx 180 ry 0 rz 0 deg; joints [-3.636, -51.481, 151.629, -3.687, -99.258, -0.377] to (266.79, -422.22, -4.17) mm, rotated rx -180 ry 0 rz 0 deg; joints [-3.637, -51.461, 151.656, -3.69, -99.304, -0.38]
  Set speed (50.8 mm/s)
  MoveL 732 to (267.42, -422.22, -4.18) mm, rotated rx -180 ry 0 rz 0 deg; joints [-3.64, -51.462, 151.699, -3.693, -99.347, -0.384]
  MoveC 733 to (267.87, -422.41, -4.18) mm, rotated rx -180 ry 0 rz 0 deg; joints [-3.654, -51.462, 151.729, -3.707, -99.376, -0.388] to (268.06, -422.86, -4.18) mm, rotated rx -180 ry 0 rz 0 deg; joints [-3.684, -51.462, 151.74, -3.738, -99.387, -0.394]
  MoveL 734 to (268.06, -448.26, -4.18) mm, rotated rx -180 ry 0 rz 0 deg; joints [-5.339, -51.45, 151.6, -5.412, -99.236, -0.68]
  MoveL 735 to (217.26, -448.26, -4.17) mm, rotated rx 180 ry 0 rz 0 deg; joints [-5.047, -51.228, 148.073, -5.078, -95.949, -0.332]
  MoveL 736 to (217.26, -397.46, -4.17) mm, rotated rx -180 ry 0 rz 0 deg; joints [-1.912, -51.27, 148.294, -1.927, -96.151, 0.037]
  MoveL 737 to (268.06, -397.46, -4.18) mm, rotated rx -180 ry 0 rz 0 deg; joints [-2.024, -51.475, 151.83, -2.055, -99.479, -0.097]
  MoveL 738 to (268.06, -422.86, -4.18) mm, rotated rx -180 ry 0 rz 0 deg; joints [-3.684, -51.462, 151.74, -3.738, -99.387, -0.394]
  MoveC 739 to (267.87, -423.31, -4.18) mm, rotated rx -180 ry 0 rz 0 deg; joints [-3.713, -51.462, 151.725, -3.767, -99.372, -0.398] to (267.42, -423.49, -4.18) mm, rotated rx -180 ry 0 rz 0 deg; joints [-3.723, -51.461, 151.694, -3.777, -99.341, -0.398]
  MoveL 740 to (266.79, -423.49, -4.17) mm, rotated rx 180 ry 0 rz 0 deg; joints [-3.72, -51.461, 151.65, -3.774, -99.298, -0.395]
  MoveC 741 to (266.34, -423.49, -3.99) mm, rotated rx -180 ry 0 rz 0 deg; joints [-3.718, -51.48, 151.623, -3.771, -99.252, -0.391] to (266.15, -423.49, -3.54) mm, rotated rx 180 ry 0 rz 0 deg; joints [-3.718, -51.529, 151.619, -3.77, -99.2, -0.388]
  Set speed (500.0 mm/s)
  MoveL 742 to (266.15, -423.49, 5) mm, rotated rx 180 ry 0 rz 0 deg; joints [-3.72, -52.457, 151.792, -3.764, -98.446, -0.338]
  MoveL 743 to (266.15, -422.22, 5) mm, rotated rx 180 ry 0 rz 0 deg; joints [-3.637, -52.457, 151.798, -3.681, -98.452, -0.325]
  Set speed (25.4 mm/s)
  MoveL 744 to (266.15, -422.22, 1.82) mm, rotated rx -180 ry 0 rz 0 deg; joints [-3.636, -52.112, 151.734, -3.683, -98.733, -0.343]
  MoveL 745 to (266.15, -422.22, -7.72) mm, rotated rx 180 ry 0 rz 0 deg; joints [-3.634, -51.077, 151.537, -3.689, -99.57, -0.397]
  MoveC 746 to (266.34, -422.22, -8.16) mm, rotated rx -180 ry 0 rz 0 deg; joints [-3.635, -51.028, 151.541, -3.69, -99.622, -0.401] to (266.79, -422.22, -8.35) mm, rotated rx -180 ry 0 rz 0 deg; joints [-3.636, -51.008, 151.568, -3.693, -99.668, -0.404]
  Set speed (50.8 mm/s)
  MoveL 747 to (267.42, -422.22, -8.35) mm, rotated rx -180 ry 0 rz 0 deg; joints [-3.639, -51.009, 151.611, -3.696, -99.711, -0.407]
  MoveC 748 to (267.87, -422.41, -8.35) mm, rotated rx -180 ry 0 rz 0 deg; joints [-3.653, -51.009, 151.641, -3.71, -99.741, -0.412] to (268.06, -422.86, -8.35) mm, rotated rx -180 ry 0 rz 0 deg; joints [-3.683, -51.009, 151.652, -3.741, -99.752, -0.418]
  MoveL 749 to (268.06, -448.26, -8.35) mm, rotated rx 180 ry 0 rz 0 deg; joints [-5.338, -50.998, 151.512, -5.417, -99.599, -0.715]
  MoveL 750 to (217.26, -448.26, -8.35) mm, rotated rx 180 ry 0 rz 0 deg; joints [-5.046, -50.809, 147.991, -5.08, -96.285, -0.362]
  MoveL 751 to (217.26, -397.46, -8.35) mm, rotated rx 180 ry 0 rz 0 deg; joints [-1.911, -50.848, 148.212, -1.927, -96.49, 0.025]
  MoveL 752 to (268.06, -397.46, -8.35) mm, rotated rx -180 ry 0 rz 0 deg; joints [-2.022, -51.02, 151.742, -2.057, -99.845, -0.11]
  MoveL 753 to (268.06, -422.86, -8.35) mm, rotated rx -180 ry 0 rz 0 deg; joints [-3.683, -51.009, 151.652, -3.741, -99.752, -0.418]
  MoveC 754 to (267.87, -423.31, -8.35) mm, rotated rx -180 ry 0 rz 0 deg; joints [-3.712, -51.008, 151.637, -3.77, -99.737, -0.423] to (267.42, -423.49, -8.35) mm, rotated rx 180 ry 0 rz 0 deg; joints [-3.722, -51.008, 151.606, -3.78, -99.705, -0.422]
  MoveL 755 to (266.79, -423.49, -8.35) mm, rotated rx -180 ry 0 rz 0 deg; joints [-3.719, -51.008, 151.562, -3.776, -99.662, -0.419]
  MoveC 756 to (266.34, -423.49, -8.16) mm, rotated rx -180 ry 0 rz 0 deg; joints [-3.717, -51.028, 151.535, -3.774, -99.616, -0.416] to (266.15, -423.49, -7.72) mm, rotated rx -180 ry 0 rz 0 deg; joints [-3.717, -51.076, 151.532, -3.773, -99.564, -0.412]
  Set speed (500.0 mm/s)
  MoveL 757 to (266.15, -423.49, 6) mm, rotated rx -180 ry 0 rz 0 deg; joints [-3.72, -52.566, 151.811, -3.764, -98.357, -0.332]
  MoveL 758 to (139.15, -422.22, 6) mm, rotated rx -180 ry 0 rz 0 deg; joints [-3.177, -51.351, 142.825, -3.181, -90.603, 0.191]
  Set speed (25.4 mm/s)
  MoveL 759 to (139.15, -422.22, -3.54) mm, rotated rx -180 ry 0 rz 0 deg; joints [-3.175, -50.487, 142.663, -3.18, -91.304, 0.152]
  MoveC 760 to (139.34, -422.22, -3.99) mm, rotated rx -180 ry 0 rz 0 deg; joints [-3.176, -50.448, 142.669, -3.18, -91.347, 0.149] to (139.79, -422.22, -4.17) mm, rotated rx -180 ry 0 rz 0 deg; joints [-3.177, -50.438, 142.698, -3.182, -91.387, 0.147]
  Set speed (50.8 mm/s)
  MoveL 761 to (140.42, -422.22, -4.18) mm, rotated rx -180 ry 0 rz 0 deg; joints [-3.179, -50.446, 142.744, -3.184, -91.424, 0.145]
  MoveC 762 to (140.87, -422.41, -4.17) mm, rotated rx -180 ry 0 rz 0 deg; joints [-3.191, -50.452, 142.775, -3.196, -91.45, 0.143] to (141.06, -422.86, -4.18) mm, rotated rx 180 ry 0 rz 0 deg; joints [-3.217, -50.454, 142.787, -3.222, -91.459, 0.141]
  MoveL 763 to (141.06, -448.26, -4.18) mm, rotated rx -180 ry 0 rz 0 deg; joints [-4.664, -50.422, 142.659, -4.669, -91.36, 0.09]
  MoveL 764 to (90.26, -448.26, -4.17) mm, rotated rx 180 ry 0 rz 0 deg; joints [-4.44, -49.63, 138.965, -4.445, -88.467, 0.324]
  MoveL 765 to (90.26, -397.46, -4.17) mm, rotated rx 180 ry 0 rz 0 deg; joints [-1.681, -49.694, 139.168, -1.685, -88.604, 0.288]
  MoveL 766 to (141.06, -397.46, -4.17) mm, rotated rx -180 ry 0 rz 0 deg; joints [-1.766, -50.479, 142.869, -1.771, -91.519, 0.199]
  MoveL 767 to (141.06, -422.86, -4.18) mm, rotated rx 180 ry 0 rz 0 deg; joints [-3.217, -50.454, 142.787, -3.222, -91.459, 0.141]
  MoveC 768 to (140.87, -423.31, -4.17) mm, rotated rx 180 ry 0 rz 0 deg; joints [-3.242, -50.451, 142.772, -3.247, -91.447, 0.141] to (140.42, -423.49, -4.17) mm, rotated rx -180 ry 0 rz 0 deg; joints [-3.251, -50.445, 142.738, -3.256, -91.42, 0.142]
  MoveL 769 to (139.79, -423.49, -4.18) mm, rotated rx 180 ry 0 rz 0 deg; joints [-3.249, -50.436, 142.693, -3.254, -91.383, 0.144]
  MoveC 770 to (139.34, -423.49, -3.99) mm, rotated rx 180 ry 0 rz 0 deg; joints [-3.248, -50.447, 142.663, -3.253, -91.343, 0.147] to (139.15, -423.49, -3.54) mm, rotated rx -180 ry 0 rz 0 deg; joints [-3.248, -50.485, 142.658, -3.252, -91.3, 0.149]
  Set speed (500.0 mm/s)
  MoveL 771 to (139.15, -423.49, 5) mm, rotated rx 180 ry 0 rz 0 deg; joints [-3.249, -51.259, 142.803, -3.253, -90.673, 0.185]
  MoveL 772 to (139.15, -422.22, 5) mm, rotated rx -180 ry 0 rz 0 deg; joints [-3.177, -51.26, 142.809, -3.181, -90.677, 0.186]
  Set speed (25.4 mm/s)
  MoveL 773 to (139.15, -422.22, 1.83) mm, rotated rx -180 ry 0 rz 0 deg; joints [-3.176, -50.972, 142.755, -3.181, -90.911, 0.173]
  MoveL 774 to (139.15, -422.22, -7.71) mm, rotated rx -180 ry 0 rz 0 deg; joints [-3.174, -50.109, 142.589, -3.179, -91.607, 0.135]
  MoveC 775 to (139.34, -422.22, -8.16) mm, rotated rx -180 ry 0 rz 0 deg; joints [-3.175, -50.07, 142.594, -3.18, -91.651, 0.132] to (139.79, -422.22, -8.35) mm, rotated rx -180 ry 0 rz 0 deg; joints [-3.176, -50.059, 142.624, -3.181, -91.691, 0.13]
  Set speed (50.8 mm/s)
  MoveL 776 to (140.42, -422.22, -8.35) mm, rotated rx 180 ry 0 rz 0 deg; joints [-3.178, -50.068, 142.669, -3.183, -91.728, 0.128]
  MoveC 777 to (140.87, -422.41, -8.35) mm, rotated rx -180 ry 0 rz 0 deg; joints [-3.19, -50.074, 142.701, -3.195, -91.754, 0.126] to (141.06, -422.86, -8.35) mm, rotated rx -180 ry 0 rz 0 deg; joints [-3.216, -50.076, 142.712, -3.222, -91.763, 0.124]
  MoveL 778 to (141.06, -448.26, -8.35) mm, rotated rx -180 ry 0 rz 0 deg; joints [-4.663, -50.044, 142.585, -4.669, -91.663, 0.066]
  MoveL 779 to (90.26, -448.26, -8.35) mm, rotated rx 180 ry 0 rz 0 deg; joints [-4.439, -49.276, 138.894, -4.443, -88.75, 0.302]
  MoveL 780 to (90.26, -397.46, -8.35) mm, rotated rx -180 ry 0 rz 0 deg; joints [-1.68, -49.339, 139.097, -1.684, -88.889, 0.279]
  MoveL 781 to (141.06, -397.46, -8.35) mm, rotated rx -180 ry 0 rz 0 deg; joints [-1.765, -50.099, 142.794, -1.77, -91.824, 0.189]
  MoveL 782 to (141.06, -422.86, -8.35) mm, rotated rx -180 ry 0 rz 0 deg; joints [-3.216, -50.076, 142.712, -3.222, -91.763, 0.124]
  MoveC 783 to (140.87, -423.31, -8.35) mm, rotated rx -180 ry 0 rz 0 deg; joints [-3.241, -50.073, 142.697, -3.247, -91.751, 0.124] to (140.42, -423.49, -8.35) mm, rotated rx 180 ry 0 rz 0 deg; joints [-3.251, -50.066, 142.664, -3.256, -91.724, 0.125]
  MoveL 784 to (139.79, -423.49, -8.35) mm, rotated rx 180 ry 0 rz 0 deg; joints [-3.249, -50.058, 142.618, -3.254, -91.687, 0.127]
  MoveC 785 to (139.34, -423.49, -8.16) mm, rotated rx -180 ry 0 rz 0 deg; joints [-3.247, -50.069, 142.589, -3.252, -91.647, 0.129] to (139.15, -423.49, -7.72) mm, rotated rx -180 ry 0 rz 0 deg; joints [-3.247, -50.107, 142.584, -3.252, -91.603, 0.132]
  Set speed (500.0 mm/s)
  MoveL 786 to (139.15, -423.49, 6) mm, rotated rx -180 ry 0 rz 0 deg; joints [-3.25, -51.349, 142.82, -3.254, -90.599, 0.189]
  MoveL 787 to (-92.16, -422.22, 6) mm, rotated rx 180 ry 0 rz 0 deg; joints [-2.582, -46.282, 125.321, -2.642, -78.181, 0.775]
  Set speed (25.4 mm/s)
  MoveL 788 to (-92.16, -422.22, -3.54) mm, rotated rx -180 ry 0 rz 0 deg; joints [-2.58, -45.621, 125.189, -2.635, -78.709, 0.749]
  MoveC 789 to (-91.98, -422.22, -3.99) mm, rotated rx -180 ry 0 rz 0 deg; joints [-2.581, -45.595, 125.197, -2.635, -78.744, 0.748] to (-91.53, -422.22, -4.17) mm, rotated rx 180 ry 0 rz 0 deg; joints [-2.582, -45.594, 125.23, -2.636, -78.778, 0.746]
  Set speed (50.8 mm/s)
  MoveL 790 to (-90.89, -422.22, -4.17) mm, rotated rx -180 ry 0 rz 0 deg; joints [-2.583, -45.611, 125.281, -2.637, -78.811, 0.745]
  MoveC 791 to (-90.44, -422.41, -4.18) mm, rotated rx -180 ry 0 rz 0 deg; joints [-2.592, -45.623, 125.316, -2.646, -78.834, 0.746] to (-90.26, -422.86, -4.18) mm, rotated rx -180 ry 0 rz 0 deg; joints [-2.614, -45.627, 125.329, -2.668, -78.843, 0.749]
  MoveL 792 to (-90.26, -448.26, -4.17) mm, rotated rx 180 ry 0 rz 0 deg; joints [-3.791, -45.582, 125.215, -3.868, -78.786, 0.968]
  MoveL 793 to (-141.06, -448.26, -4.17) mm, rotated rx 180 ry 0 rz 0 deg; joints [-3.641, -44.155, 121.139, -3.754, -76.142, 1.117]
  MoveL 794 to (-141.06, -397.46, -4.17) mm, rotated rx -180 ry 0 rz 0 deg; joints [-1.377, -44.233, 121.323, -1.422, -76.224, 0.59]
  MoveL 795 to (-90.26, -397.46, -4.17) mm, rotated rx 180 ry 0 rz 0 deg; joints [-1.434, -45.659, 125.402, -1.466, -78.876, 0.533]
  MoveL 796 to (-90.26, -422.86, -4.18) mm, rotated rx -180 ry 0 rz 0 deg; joints [-2.614, -45.627, 125.329, -2.668, -78.843, 0.749]
  MoveC 797 to (-90.44, -423.31, -4.18) mm, rotated rx -180 ry 0 rz 0 deg; joints [-2.634, -45.622, 125.312, -2.689, -78.832, 0.753] to (-90.89, -423.49, -4.18) mm, rotated rx -180 ry 0 rz 0 deg; joints [-2.642, -45.609, 125.276, -2.697, -78.808, 0.756]
  MoveL 798 to (-91.53, -423.49, -4.18) mm, rotated rx 180 ry 0 rz 0 deg; joints [-2.64, -45.592, 125.226, -2.696, -78.775, 0.757]
  MoveC 799 to (-91.98, -423.49, -3.99) mm, rotated rx -180 ry 0 rz 0 deg; joints [-2.64, -45.593, 125.193, -2.695, -78.742, 0.759] to (-92.16, -423.49, -3.54) mm, rotated rx 180 ry 0 rz 0 deg; joints [-2.639, -45.619, 125.184, -2.695, -78.707, 0.76]
  Set speed (500.0 mm/s)
  MoveL 800 to (-92.16, -423.49, 5) mm, rotated rx -180 ry 0 rz 0 deg; joints [-2.641, -46.211, 125.303, -2.701, -78.234, 0.783]
  MoveL 801 to (-92.16, -422.22, 5) mm, rotated rx -180 ry 0 rz 0 deg; joints [-2.582, -46.213, 125.307, -2.641, -78.236, 0.772]
  Set speed (25.4 mm/s)
  MoveL 802 to (-92.16, -422.22, 1.82) mm, rotated rx 180 ry 0 rz 0 deg; joints [-2.581, -45.993, 125.264, -2.639, -78.413, 0.764]
  MoveL 803 to (-92.16, -422.22, -7.71) mm, rotated rx -180 ry 0 rz 0 deg; joints [-2.58, -45.331, 125.129, -2.632, -78.939, 0.738]
  MoveC 804 to (-91.98, -422.22, -8.16) mm, rotated rx 180 ry 0 rz 0 deg; joints [-2.58, -45.305, 125.137, -2.632, -78.973, 0.737] to (-91.53, -422.22, -8.35) mm, rotated rx 180 ry 0 rz 0 deg; joints [-2.581, -45.304, 125.17, -2.633, -79.007, 0.736]
  Set speed (50.8 mm/s)
  MoveL 805 to (-90.89, -422.22, -8.35) mm, rotated rx 180 ry 0 rz 0 deg; joints [-2.582, -45.321, 125.22, -2.634, -79.04, 0.734]
  MoveC 806 to (-90.44, -422.41, -8.35) mm, rotated rx -180 ry 0 rz 0 deg; joints [-2.592, -45.333, 125.255, -2.644, -79.063, 0.735] to (-90.26, -422.86, -8.35) mm, rotated rx -180 ry 0 rz 0 deg; joints [-2.613, -45.337, 125.268, -2.665, -79.072, 0.738]
  MoveL 807 to (-90.26, -448.26, -8.35) mm, rotated rx 180 ry 0 rz 0 deg; joints [-3.79, -45.292, 125.154, -3.865, -79.015, 0.952]
  MoveL 808 to (-141.06, -448.26, -8.35) mm, rotated rx -180 ry 0 rz 0 deg; joints [-3.64, -43.879, 121.081, -3.75, -76.359, 1.103]
  MoveL 809 to (-141.06, -397.46, -8.35) mm, rotated rx 180 ry 0 rz 0 deg; joints [-1.377, -43.957, 121.265, -1.42, -76.442, 0.584]
  MoveL 810 to (-90.26, -397.46, -8.35) mm, rotated rx 180 ry 0 rz 0 deg; joints [-1.433, -45.368, 125.341, -1.464, -79.106, 0.527]
  MoveL 811 to (-90.26, -422.86, -8.35) mm, rotated rx -180 ry 0 rz 0 deg; joints [-2.613, -45.337, 125.268, -2.665, -79.072, 0.738]
  MoveC 812 to (-90.44, -423.31, -8.35) mm, rotated rx -180 ry 0 rz 0 deg; joints [-2.633, -45.331, 125.252, -2.686, -79.062, 0.742] to (-90.89, -423.49, -8.35) mm, rotated rx -180 ry 0 rz 0 deg; joints [-2.641, -45.319, 125.216, -2.694, -79.038, 0.745]
  MoveL 813 to (-91.53, -423.49, -8.35) mm, rotated rx -180 ry 0 rz 0 deg; joints [-2.64, -45.302, 125.165, -2.693, -79.005, 0.746]
  MoveC 814 to (-91.98, -423.49, -8.16) mm, rotated rx -180 ry 0 rz 0 deg; joints [-2.639, -45.303, 125.133, -2.692, -78.971, 0.748] to (-92.16, -423.49, -7.72) mm, rotated rx 180 ry 0 rz 0 deg; joints [-2.638, -45.329, 125.124, -2.692, -78.936, 0.749]
  Set speed (500.0 mm/s)
  MoveL 815 to (-92.16, -423.49, 6) mm, rotated rx -180 ry 0 rz 0 deg; joints [-2.641, -46.28, 125.316, -2.702, -78.179, 0.786]
  MoveL 816 to (-219.16, -422.22, 6) mm, rotated rx 180 ry 0 rz 0 deg; joints [-2.341, -42.413, 114.901, -2.471, -71.633, 1.016]
  Set speed (25.4 mm/s)
  MoveL 817 to (-219.16, -422.22, -3.54) mm, rotated rx -180 ry 0 rz 0 deg; joints [-2.34, -41.827, 114.777, -2.463, -72.096, 0.994]
  MoveC 818 to (-218.98, -422.22, -3.99) mm, rotated rx -180 ry 0 rz 0 deg; joints [-2.34, -41.805, 114.787, -2.463, -72.127, 0.993] to (-218.53, -422.22, -4.17) mm, rotated rx 180 ry 0 rz 0 deg; joints [-2.341, -41.809, 114.823, -2.463, -72.16, 0.992]
  Set speed (50.8 mm/s)
  MoveL 819 to (-217.89, -422.22, -4.18) mm, rotated rx -180 ry 0 rz 0 deg; joints [-2.342, -41.829, 114.877, -2.464, -72.193, 0.991]
  MoveC 820 to (-217.44, -422.41, -4.18) mm, rotated rx 180 ry 0 rz 0 deg; joints [-2.35, -41.844, 114.914, -2.472, -72.216, 0.992] to (-217.26, -422.86, -4.18) mm, rotated rx -180 ry 0 rz 0 deg; joints [-2.369, -41.849, 114.928, -2.492, -72.225, 0.998]
  MoveL 821 to (-217.26, -448.26, -4.18) mm, rotated rx -180 ry 0 rz 0 deg; joints [-3.437, -41.801, 114.818, -3.615, -72.179, 1.328]
  MoveL 822 to (-268.06, -448.26, -4.18) mm, rotated rx -180 ry 0 rz 0 deg; joints [-3.314, -40.091, 110.443, -3.541, -69.517, 1.463]
  MoveL 823 to (-268.06, -397.46, -4.18) mm, rotated rx 180 ry 0 rz 0 deg; joints [-1.253, -40.174, 110.624, -1.341, -69.585, 0.721]
  MoveL 824 to (-217.26, -397.46, -4.18) mm, rotated rx 180 ry 0 rz 0 deg; joints [-1.3, -41.882, 114.999, -1.369, -72.252, 0.67]
  MoveL 825 to (-217.26, -422.86, -4.18) mm, rotated rx -180 ry 0 rz 0 deg; joints [-2.369, -41.849, 114.928, -2.492, -72.225, 0.998]
  MoveC 826 to (-217.44, -423.31, -4.18) mm, rotated rx -180 ry 0 rz 0 deg; joints [-2.388, -41.842, 114.911, -2.512, -72.215, 1.004] to (-217.89, -423.49, -4.17) mm, rotated rx -180 ry 0 rz 0 deg; joints [-2.395, -41.827, 114.872, -2.52, -72.191, 1.007]
  MoveL 827 to (-218.53, -423.49, -4.18) mm, rotated rx 180 ry 0 rz 0 deg; joints [-2.394, -41.806, 114.818, -2.519, -72.158, 1.008]
  MoveC 828 to (-218.98, -423.49, -3.99) mm, rotated rx -180 ry 0 rz 0 deg; joints [-2.393, -41.803, 114.783, -2.519, -72.125, 1.009] to (-219.16, -423.49, -3.54) mm, rotated rx 180 ry 0 rz 0 deg; joints [-2.393, -41.825, 114.773, -2.519, -72.094, 1.011]
  Set speed (500.0 mm/s)
  MoveL 829 to (-219.16, -423.49, 5) mm, rotated rx -180 ry 0 rz 0 deg; joints [-2.394, -42.35, 114.884, -2.526, -71.68, 1.03]
  MoveL 830 to (-219.16, -422.22, 5) mm, rotated rx -180 ry 0 rz 0 deg; joints [-2.341, -42.352, 114.888, -2.47, -71.682, 1.014]
  Set speed (25.4 mm/s)
  MoveL 831 to (-219.16, -422.22, 1.83) mm, rotated rx -180 ry 0 rz 0 deg; joints [-2.34, -42.157, 114.848, -2.467, -71.836, 1.006]
  MoveL 832 to (-219.16, -422.22, -7.71) mm, rotated rx -180 ry 0 rz 0 deg; joints [-2.339, -41.57, 114.721, -2.459, -72.297, 0.985]
  MoveC 833 to (-218.98, -422.22, -8.16) mm, rotated rx 180 ry 0 rz 0 deg; joints [-2.339, -41.548, 114.731, -2.459, -72.328, 0.984] to (-218.53, -422.22, -8.35) mm, rotated rx -180 ry 0 rz 0 deg; joints [-2.34, -41.551, 114.766, -2.459, -72.36, 0.982]
  Set speed (50.8 mm/s)
  MoveL 834 to (-217.89, -422.22, -8.35) mm, rotated rx 180 ry 0 rz 0 deg; joints [-2.341, -41.572, 114.82, -2.46, -72.394, 0.981]
  MoveC 835 to (-217.44, -422.41, -8.35) mm, rotated rx -180 ry 0 rz 0 deg; joints [-2.35, -41.586, 114.858, -2.469, -72.417, 0.983] to (-217.26, -422.86, -8.35) mm, rotated rx -180 ry 0 rz 0 deg; joints [-2.369, -41.591, 114.872, -2.489, -72.426, 0.988]
  MoveL 836 to (-217.26, -448.26, -8.35) mm, rotated rx -180 ry 0 rz 0 deg; joints [-3.437, -41.543, 114.761, -3.61, -72.38, 1.314]
  MoveL 837 to (-268.06, -448.26, -8.35) mm, rotated rx 180 ry 0 rz 0 deg; joints [-3.313, -39.844, 110.388, -3.536, -69.708, 1.45]
  MoveL 838 to (-268.06, -397.46, -8.35) mm, rotated rx 180 ry 0 rz 0 deg; joints [-1.252, -39.927, 110.568, -1.339, -69.776, 0.716]
  MoveL 839 to (-217.26, -397.46, -8.35) mm, rotated rx -180 ry 0 rz 0 deg; joints [-1.299, -41.624, 114.942, -1.367, -72.453, 0.665]
  MoveL 840 to (-217.26, -422.86, -8.35) mm, rotated rx -180 ry 0 rz 0 deg; joints [-2.369, -41.591, 114.872, -2.489, -72.426, 0.988]
  MoveC 841 to (-217.44, -423.31, -8.35) mm, rotated rx -180 ry 0 rz 0 deg; joints [-2.387, -41.584, 114.854, -2.508, -72.416, 0.994] to (-217.89, -423.49, -8.35) mm, rotated rx 180 ry 0 rz 0 deg; joints [-2.394, -41.57, 114.816, -2.516, -72.392, 0.998]
  MoveL 842 to (-218.53, -423.49, -8.35) mm, rotated rx -180 ry 0 rz 0 deg; joints [-2.393, -41.549, 114.762, -2.515, -72.359, 0.999]
  MoveC 843 to (-218.98, -423.49, -8.16) mm, rotated rx -180 ry 0 rz 0 deg; joints [-2.392, -41.546, 114.726, -2.515, -72.326, 1] to (-219.16, -423.49, -7.72) mm, rotated rx -180 ry 0 rz 0 deg; joints [-2.392, -41.568, 114.717, -2.515, -72.295, 1.001]
  Set speed (500.0 mm/s)
  MoveL 844 to (-219.16, -423.49, 6) mm, rotated rx 180 ry 0 rz 0 deg; joints [-2.395, -42.411, 114.896, -2.527, -71.631, 1.033]
  MoveL 845 to (-346.16, -422.22, 6) mm, rotated rx -180 ry 0 rz 0 deg; joints [-2.141, -37.851, 103.659, -2.368, -64.956, 1.243]
  Set speed (25.4 mm/s)
  MoveL 846 to (-346.16, -422.22, -3.54) mm, rotated rx -180 ry 0 rz 0 deg; joints [-2.14, -37.323, 103.539, -2.358, -65.365, 1.223]
  MoveC 847 to (-345.98, -422.22, -3.99) mm, rotated rx -180 ry 0 rz 0 deg; joints [-2.14, -37.305, 103.551, -2.358, -65.394, 1.222] to (-345.53, -422.22, -4.17) mm, rotated rx -180 ry 0 rz 0 deg; joints [-2.141, -37.312, 103.59, -2.358, -65.426, 1.221]
  Set speed (50.8 mm/s)
  MoveL 848 to (-344.89, -422.22, -4.18) mm, rotated rx 180 ry 0 rz 0 deg; joints [-2.142, -37.336, 103.649, -2.359, -65.46, 1.22]
  MoveC 849 to (-344.44, -422.41, -4.18) mm, rotated rx 180 ry 0 rz 0 deg; joints [-2.149, -37.353, 103.689, -2.367, -65.485, 1.222] to (-344.26, -422.86, -4.18) mm, rotated rx -180 ry 0 rz 0 deg; joints [-2.167, -37.359, 103.705, -2.386, -65.494, 1.229]
  MoveL 850 to (-344.26, -448.26, -4.17) mm, rotated rx 180 ry 0 rz 0 deg; joints [-3.144, -37.309, 103.595, -3.461, -65.455, 1.664]
  MoveL 851 to (-395.06, -448.26, -4.18) mm, rotated rx -180 ry 0 rz 0 deg; joints [-3.04, -35.298, 98.802, -3.427, -62.675, 1.8]
  MoveL 852 to (-395.06, -397.46, -4.18) mm, rotated rx -180 ry 0 rz 0 deg; joints [-1.149, -35.386, 98.984, -1.297, -62.735, 0.849]
  MoveL 853 to (-344.26, -397.46, -4.17) mm, rotated rx -180 ry 0 rz 0 deg; joints [-1.189, -37.394, 103.775, -1.31, -65.517, 0.797]
  MoveL 854 to (-344.26, -422.86, -4.18) mm, rotated rx -180 ry 0 rz 0 deg; joints [-2.167, -37.359, 103.705, -2.386, -65.494, 1.229]
  MoveC 855 to (-344.44, -423.31, -4.18) mm, rotated rx 180 ry 0 rz 0 deg; joints [-2.184, -37.352, 103.686, -2.405, -65.483, 1.237] to (-344.89, -423.49, -4.17) mm, rotated rx -180 ry 0 rz 0 deg; joints [-2.19, -37.334, 103.644, -2.412, -65.459, 1.241]
  MoveL 856 to (-345.53, -423.49, -4.18) mm, rotated rx 180 ry 0 rz 0 deg; joints [-2.189, -37.31, 103.585, -2.412, -65.425, 1.243]
  MoveC 857 to (-345.98, -423.49, -3.99) mm, rotated rx -180 ry 0 rz 0 deg; joints [-2.189, -37.303, 103.546, -2.412, -65.392, 1.244] to (-346.16, -423.49, -3.54) mm, rotated rx 180 ry 0 rz 0 deg; joints [-2.189, -37.321, 103.535, -2.412, -65.363, 1.245]
  Set speed (500.0 mm/s)
  MoveL 858 to (-346.16, -423.49, 5) mm, rotated rx -180 ry 0 rz 0 deg; joints [-2.19, -37.794, 103.642, -2.421, -64.998, 1.263]
  MoveL 859 to (-346.16, -422.22, 5) mm, rotated rx -180 ry 0 rz 0 deg; joints [-2.141, -37.796, 103.646, -2.367, -64.999, 1.241]
  Set speed (25.4 mm/s)
  MoveL 860 to (-346.16, -422.22, 1.83) mm, rotated rx -180 ry 0 rz 0 deg; joints [-2.141, -37.62, 103.607, -2.364, -65.135, 1.234]
  MoveL 861 to (-346.16, -422.22, -7.72) mm, rotated rx 180 ry 0 rz 0 deg; joints [-2.139, -37.091, 103.485, -2.354, -65.542, 1.215]
  MoveC 862 to (-345.98, -422.22, -8.16) mm, rotated rx 180 ry 0 rz 0 deg; joints [-2.139, -37.073, 103.496, -2.354, -65.571, 1.214] to (-345.53, -422.22, -8.35) mm, rotated rx -180 ry 0 rz 0 deg; joints [-2.14, -37.08, 103.535, -2.354, -65.603, 1.213]
  Set speed (50.8 mm/s)
  MoveL 863 to (-344.89, -422.22, -8.35) mm, rotated rx -180 ry 0 rz 0 deg; joints [-2.141, -37.104, 103.594, -2.354, -65.638, 1.211]
  MoveC 864 to (-344.44, -422.41, -8.35) mm, rotated rx -180 ry 0 rz 0 deg; joints [-2.149, -37.121, 103.635, -2.363, -65.662, 1.214] to (-344.26, -422.86, -8.35) mm, rotated rx 180 ry 0 rz 0 deg; joints [-2.166, -37.127, 103.65, -2.382, -65.672, 1.221]
  MoveL 865 to (-344.26, -448.26, -8.35) mm, rotated rx -180 ry 0 rz 0 deg; joints [-3.143, -37.076, 103.54, -3.455, -65.632, 1.652]
  MoveL 866 to (-395.06, -448.26, -8.35) mm, rotated rx -180 ry 0 rz 0 deg; joints [-3.039, -35.074, 98.748, -3.421, -62.844, 1.789]
  MoveL 867 to (-395.06, -397.46, -8.35) mm, rotated rx 180 ry 0 rz 0 deg; joints [-1.149, -35.161, 98.93, -1.295, -62.904, 0.845]
  MoveL 868 to (-344.26, -397.46, -8.35) mm, rotated rx 180 ry 0 rz 0 deg; joints [-1.188, -37.162, 103.721, -1.308, -65.695, 0.793]
  MoveL 869 to (-344.26, -422.86, -8.35) mm, rotated rx 180 ry 0 rz 0 deg; joints [-2.166, -37.127, 103.65, -2.382, -65.672, 1.221]
  MoveC 870 to (-344.44, -423.31, -8.35) mm, rotated rx -180 ry 0 rz 0 deg; joints [-2.183, -37.119, 103.631, -2.401, -65.661, 1.229] to (-344.89, -423.49, -8.35) mm, rotated rx -180 ry 0 rz 0 deg; joints [-2.19, -37.102, 103.589, -2.408, -65.636, 1.233]
  MoveL 871 to (-345.53, -423.49, -8.35) mm, rotated rx 180 ry 0 rz 0 deg; joints [-2.189, -37.078, 103.53, -2.408, -65.602, 1.234]
  MoveC 872 to (-345.98, -423.49, -8.16) mm, rotated rx -180 ry 0 rz 0 deg; joints [-2.188, -37.071, 103.491, -2.408, -65.57, 1.235] to (-346.16, -423.49, -7.72) mm, rotated rx -180 ry 0 rz 0 deg; joints [-2.188, -37.089, 103.48, -2.408, -65.54, 1.237]
  Set speed (500.0 mm/s)
  MoveL 873 to (-346.16, -423.49, 6) mm, rotated rx -180 ry 0 rz 0 deg; joints [-2.19, -37.849, 103.654, -2.422, -64.954, 1.265]
  MoveL 874 to (-346.16, -235.88, 6) mm, rotated rx -180 ry 0 rz 0 deg; joints [5.018, -37.722, 103.237, 5.544, -64.746, -2.023]
  Set speed (25.4 mm/s)
  MoveL 875 to (-346.16, -235.89, -3.54) mm, rotated rx 180 ry 0 rz 0 deg; joints [5.02, -37.195, 103.118, 5.528, -65.151, -1.98]
  MoveC 876 to (-345.98, -235.88, -3.99) mm, rotated rx -180 ry 0 rz 0 deg; joints [5.021, -37.178, 103.129, 5.528, -65.18, -1.978] to (-345.53, -235.89, -4.17) mm, rotated rx -180 ry 0 rz 0 deg; joints [5.022, -37.185, 103.168, 5.528, -65.212, -1.975]
  Set speed (50.8 mm/s)
  MoveL 877 to (-344.89, -235.88, -4.17) mm, rotated rx -180 ry 0 rz 0 deg; joints [5.024, -37.209, 103.227, 5.529, -65.247, -1.972]
  MoveC 878 to (-344.44, -236.07, -4.17) mm, rotated rx -180 ry 0 rz 0 deg; joints [5.019, -37.227, 103.27, 5.522, -65.271, -1.967] to (-344.26, -236.52, -4.18) mm, rotated rx -180 ry 0 rz 0 deg; joints [5.002, -37.236, 103.291, 5.503, -65.283, -1.958]
  MoveL 879 to (-344.26, -261.92, -4.17) mm, rotated rx -180 ry 0 rz 0 deg; joints [4.029, -37.304, 103.474, 4.428, -65.363, -1.516]
  MoveL 880 to (-395.06, -261.92, -4.18) mm, rotated rx 180 ry 0 rz 0 deg; joints [3.897, -35.29, 98.681, 4.385, -62.588, -1.691]
  MoveL 881 to (-395.06, -211.12, -4.17) mm, rotated rx 180 ry 0 rz 0 deg; joints [5.776, -35.13, 98.27, 6.515, -62.419, -2.666]
  MoveL 882 to (-344.26, -211.12, -4.18) mm, rotated rx -180 ry 0 rz 0 deg; joints [5.972, -37.15, 103.067, 6.577, -65.187, -2.407]
  MoveL 883 to (-344.26, -236.52, -4.18) mm, rotated rx -180 ry 0 rz 0 deg; joints [5.002, -37.236, 103.291, 5.503, -65.283, -1.958]
  MoveC 884 to (-344.44, -236.97, -4.18) mm, rotated rx 180 ry 0 rz 0 deg; joints [4.984, -37.23, 103.277, 5.484, -65.275, -1.951] to (-344.89, -237.16, -4.17) mm, rotated rx -180 ry 0 rz 0 deg; joints [4.976, -37.213, 103.237, 5.475, -65.251, -1.95]
  MoveL 885 to (-345.53, -237.16, -4.18) mm, rotated rx -180 ry 0 rz 0 deg; joints [4.974, -37.189, 103.178, 5.474, -65.217, -1.953]
  MoveC 886 to (-345.98, -237.16, -3.99) mm, rotated rx 180 ry 0 rz 0 deg; joints [4.972, -37.182, 103.139, 5.474, -65.185, -1.955] to (-346.16, -237.16, -3.54) mm, rotated rx -180 ry 0 rz 0 deg; joints [4.971, -37.199, 103.128, 5.475, -65.156, -1.958]
  Set speed (500.0 mm/s)
  MoveL 887 to (-346.16, -237.16, 5) mm, rotated rx -180 ry 0 rz 0 deg; joints [4.969, -37.671, 103.235, 5.489, -64.793, -1.996]
  MoveL 888 to (-346.16, -235.88, 5) mm, rotated rx -180 ry 0 rz 0 deg; joints [5.018, -37.667, 103.225, 5.543, -64.788, -2.018]
  Set speed (25.4 mm/s)
  MoveL 889 to (-346.16, -235.89, 1.82) mm, rotated rx -180 ry 0 rz 0 deg; joints [5.019, -37.492, 103.185, 5.537, -64.924, -2.004]
  MoveL 890 to (-346.16, -235.89, -7.72) mm, rotated rx 180 ry 0 rz 0 deg; joints [5.021, -36.964, 103.063, 5.522, -65.327, -1.962]
  MoveC 891 to (-345.98, -235.88, -8.16) mm, rotated rx -180 ry 0 rz 0 deg; joints [5.022, -36.946, 103.074, 5.521, -65.356, -1.959] to (-345.53, -235.89, -8.35) mm, rotated rx -180 ry 0 rz 0 deg; joints [5.023, -36.953, 103.113, 5.521, -65.388, -1.957]
  Set speed (50.8 mm/s)
  MoveL 892 to (-344.89, -235.89, -8.35) mm, rotated rx 180 ry 0 rz 0 deg; joints [5.025, -36.978, 103.172, 5.522, -65.423, -1.954]
  MoveC 893 to (-344.44, -236.07, -8.35) mm, rotated rx 180 ry 0 rz 0 deg; joints [5.02, -36.995, 103.215, 5.515, -65.448, -1.949] to (-344.26, -236.52, -8.35) mm, rotated rx 180 ry 0 rz 0 deg; joints [5.003, -37.004, 103.236, 5.496, -65.459, -1.94]
  MoveL 894 to (-344.26, -261.92, -8.35) mm, rotated rx -180 ry 0 rz 0 deg; joints [4.03, -37.072, 103.419, 4.423, -65.54, -1.501]
  MoveL 895 to (-395.06, -261.92, -8.35) mm, rotated rx -180 ry 0 rz 0 deg; joints [3.897, -35.066, 98.626, 4.38, -62.756, -1.676]
  MoveL 896 to (-395.06, -211.12, -8.35) mm, rotated rx -180 ry 0 rz 0 deg; joints [5.777, -34.907, 98.216, 6.506, -62.586, -2.645]
  MoveL 897 to (-344.26, -211.12, -8.35) mm, rotated rx 180 ry 0 rz 0 deg; joints [5.973, -36.919, 103.013, 6.569, -65.362, -2.385]
  MoveL 898 to (-344.26, -236.52, -8.35) mm, rotated rx 180 ry 0 rz 0 deg; joints [5.003, -37.004, 103.236, 5.496, -65.459, -1.94]
  MoveC 899 to (-344.44, -236.97, -8.35) mm, rotated rx 180 ry 0 rz 0 deg; joints [4.985, -36.998, 103.222, 5.477, -65.451, -1.933] to (-344.89, -237.16, -8.35) mm, rotated rx 180 ry 0 rz 0 deg; joints [4.977, -36.981, 103.182, 5.469, -65.427, -1.932]
  MoveL 900 to (-345.53, -237.16, -8.35) mm, rotated rx -180 ry 0 rz 0 deg; joints [4.975, -36.957, 103.124, 5.468, -65.393, -1.935]
  MoveC 901 to (-345.98, -237.16, -8.16) mm, rotated rx 180 ry 0 rz 0 deg; joints [4.973, -36.95, 103.085, 5.467, -65.361, -1.937] to (-346.16, -237.15, -7.72) mm, rotated rx -180 ry 0 rz 0 deg; joints [4.972, -36.968, 103.073, 5.468, -65.332, -1.94]
  Set speed (500.0 mm/s)
  MoveL 902 to (-346.16, -237.16, 6) mm, rotated rx -180 ry 0 rz 0 deg; joints [4.969, -37.726, 103.247, 5.49, -64.75, -2]
  MoveL 903 to (-219.16, -235.88, 6) mm, rotated rx -180 ry 0 rz 0 deg; joints [5.483, -42.302, 114.478, 5.781, -71.391, -1.495]
  Set speed (25.4 mm/s)
  MoveL 904 to (-219.16, -235.88, -3.54) mm, rotated rx -180 ry 0 rz 0 deg; joints [5.485, -41.718, 114.355, 5.768, -71.85, -1.447]
  MoveC 905 to (-218.98, -235.88, -3.99) mm, rotated rx -180 ry 0 rz 0 deg; joints [5.486, -41.697, 114.365, 5.768, -71.881, -1.444] to (-218.53, -235.89, -4.17) mm, rotated rx -180 ry 0 rz 0 deg; joints [5.488, -41.7, 114.401, 5.769, -71.913, -1.441]
  Set speed (50.8 mm/s)
  MoveL 906 to (-217.89, -235.88, -4.18) mm, rotated rx -180 ry 0 rz 0 deg; joints [5.49, -41.721, 114.455, 5.771, -71.946, -1.438]
  MoveC 907 to (-217.44, -236.07, -4.18) mm, rotated rx -180 ry 0 rz 0 deg; joints [5.484, -41.736, 114.494, 5.763, -71.97, -1.434] to (-217.26, -236.52, -4.18) mm, rotated rx 180 ry 0 rz 0 deg; joints [5.466, -41.744, 114.513, 5.744, -71.981, -1.427]
  MoveL 908 to (-217.26, -261.92, -4.18) mm, rotated rx -180 ry 0 rz 0 deg; joints [4.404, -41.806, 114.697, 4.624, -72.074, -1.087]
  MoveL 909 to (-268.06, -261.92, -4.18) mm, rotated rx 180 ry 0 rz 0 deg; joints [4.246, -40.092, 110.323, 4.531, -69.418, -1.259]
  MoveL 910 to (-268.06, -211.12, -4.17) mm, rotated rx 180 ry 0 rz 0 deg; joints [6.292, -39.947, 109.917, 6.726, -69.227, -2.027]
  MoveL 911 to (-217.26, -211.12, -4.18) mm, rotated rx -180 ry 0 rz 0 deg; joints [6.525, -41.666, 114.29, 6.862, -71.871, -1.773]
  MoveL 912 to (-217.26, -236.52, -4.18) mm, rotated rx 180 ry 0 rz 0 deg; joints [5.466, -41.744, 114.513, 5.744, -71.981, -1.427]
  MoveC 913 to (-217.44, -236.97, -4.18) mm, rotated rx 180 ry 0 rz 0 deg; joints [5.447, -41.739, 114.501, 5.724, -71.974, -1.421] to (-217.89, -237.16, -4.18) mm, rotated rx 180 ry 0 rz 0 deg; joints [5.437, -41.725, 114.465, 5.715, -71.951, -1.421]
  MoveL 914 to (-218.53, -237.16, -4.18) mm, rotated rx -180 ry 0 rz 0 deg; joints [5.435, -41.704, 114.411, 5.713, -71.918, -1.424]
  MoveC 915 to (-218.98, -237.16, -3.99) mm, rotated rx -180 ry 0 rz 0 deg; joints [5.433, -41.7, 114.375, 5.712, -71.886, -1.426] to (-219.16, -237.16, -3.54) mm, rotated rx -180 ry 0 rz 0 deg; joints [5.432, -41.722, 114.365, 5.712, -71.855, -1.429]
  Set speed (500.0 mm/s)
  MoveL 916 to (-219.16, -237.16, 5) mm, rotated rx -180 ry 0 rz 0 deg; joints [5.43, -42.245, 114.476, 5.724, -71.444, -1.472]
  MoveL 917 to (-219.16, -235.88, 5) mm, rotated rx -180 ry 0 rz 0 deg; joints [5.483, -42.241, 114.466, 5.78, -71.439, -1.49]
  Set speed (25.4 mm/s)
  MoveL 918 to (-219.16, -235.88, 1.82) mm, rotated rx -180 ry 0 rz 0 deg; joints [5.484, -42.047, 114.425, 5.775, -71.592, -1.474]
  MoveL 919 to (-219.16, -235.89, -7.71) mm, rotated rx -180 ry 0 rz 0 deg; joints [5.486, -41.462, 114.299, 5.763, -72.049, -1.426]
  MoveC 920 to (-218.98, -235.88, -8.16) mm, rotated rx -180 ry 0 rz 0 deg; joints [5.487, -41.441, 114.309, 5.763, -72.08, -1.423] to (-218.53, -235.89, -8.35) mm, rotated rx -180 ry 0 rz 0 deg; joints [5.489, -41.444, 114.344, 5.764, -72.112, -1.42]
  Set speed (50.8 mm/s)
  MoveL 921 to (-217.89, -235.88, -8.35) mm, rotated rx -180 ry 0 rz 0 deg; joints [5.491, -41.465, 114.398, 5.765, -72.145, -1.417]
  MoveC 922 to (-217.44, -236.07, -8.35) mm, rotated rx -180 ry 0 rz 0 deg; joints [5.485, -41.48, 114.438, 5.758, -72.169, -1.413] to (-217.26, -236.52, -8.35) mm, rotated rx -180 ry 0 rz 0 deg; joints [5.467, -41.487, 114.457, 5.739, -72.181, -1.406]
  MoveL 923 to (-217.26, -261.92, -8.35) mm, rotated rx -180 ry 0 rz 0 deg; joints [4.405, -41.549, 114.641, 4.62, -72.274, -1.07]
  MoveL 924 to (-268.06, -261.92, -8.35) mm, rotated rx -180 ry 0 rz 0 deg; joints [4.247, -39.846, 110.267, 4.526, -69.608, -1.243]
  MoveL 925 to (-268.06, -211.12, -8.35) mm, rotated rx -180 ry 0 rz 0 deg; joints [6.293, -39.702, 109.862, 6.719, -69.416, -2.004]
  MoveL 926 to (-217.26, -211.12, -8.35) mm, rotated rx 180 ry 0 rz 0 deg; joints [6.526, -41.41, 114.233, 6.856, -72.069, -1.748]
  MoveL 927 to (-217.26, -236.52, -8.35) mm, rotated rx -180 ry 0 rz 0 deg; joints [5.467, -41.487, 114.457, 5.739, -72.181, -1.406]
  MoveC 928 to (-217.44, -236.97, -8.35) mm, rotated rx -180 ry 0 rz 0 deg; joints [5.448, -41.482, 114.445, 5.719, -72.173, -1.401] to (-217.89, -237.16, -8.35) mm, rotated rx 180 ry 0 rz 0 deg; joints [5.438, -41.468, 114.408, 5.709, -72.15, -1.4]
  MoveL 929 to (-218.53, -237.16, -8.35) mm, rotated rx -180 ry 0 rz 0 deg; joints [5.436, -41.447, 114.355, 5.708, -72.117, -1.403]
  MoveC 930 to (-218.98, -237.15, -8.16) mm, rotated rx -180 ry 0 rz 0 deg; joints [5.434, -41.444, 114.319, 5.707, -72.085, -1.406] to (-219.16, -237.16, -7.72) mm, rotated rx -180 ry 0 rz 0 deg; joints [5.433, -41.466, 114.309, 5.707, -72.054, -1.409]
  Set speed (500.0 mm/s)
  MoveL 931 to (-219.16, -237.16, 6) mm, rotated rx 180 ry 0 rz 0 deg; joints [5.43, -42.306, 114.488, 5.725, -71.396, -1.477]
  MoveL 932 to (-92.16, -235.88, 6) mm, rotated rx -180 ry 0 rz 0 deg; joints [6.042, -46.192, 124.886, 6.175, -77.888, -0.936]
  Set speed (25.4 mm/s)
  MoveL 933 to (-92.16, -235.88, -3.54) mm, rotated rx -180 ry 0 rz 0 deg; joints [6.045, -45.535, 124.755, 6.166, -78.411, -0.879]
  MoveC 934 to (-91.98, -235.89, -3.99) mm, rotated rx 180 ry 0 rz 0 deg; joints [6.046, -45.509, 124.763, 6.167, -78.445, -0.875] to (-91.53, -235.88, -4.17) mm, rotated rx -180 ry 0 rz 0 deg; joints [6.048, -45.508, 124.796, 6.168, -78.479, -0.872]
  Set speed (50.8 mm/s)
  MoveL 935 to (-90.89, -235.88, -4.17) mm, rotated rx -180 ry 0 rz 0 deg; joints [6.051, -45.525, 124.846, 6.171, -78.512, -0.869]
  MoveC 936 to (-90.44, -236.07, -4.17) mm, rotated rx 180 ry 0 rz 0 deg; joints [6.045, -45.538, 124.883, 6.164, -78.536, -0.865] to (-90.26, -236.52, -4.17) mm, rotated rx -180 ry 0 rz 0 deg; joints [6.025, -45.544, 124.902, 6.143, -78.548, -0.86]
  MoveL 937 to (-90.26, -261.92, -4.17) mm, rotated rx -180 ry 0 rz 0 deg; joints [4.855, -45.599, 125.091, 4.947, -78.661, -0.629]
  MoveL 938 to (-141.06, -261.92, -4.18) mm, rotated rx -180 ry 0 rz 0 deg; joints [4.664, -44.166, 121.017, 4.802, -76.026, -0.819]
  MoveL 939 to (-141.06, -211.12, -4.17) mm, rotated rx 180 ry 0 rz 0 deg; joints [6.909, -44.036, 120.604, 7.123, -75.798, -1.378]
  MoveL 940 to (-90.26, -211.12, -4.18) mm, rotated rx 180 ry 0 rz 0 deg; joints [7.19, -45.476, 124.672, 7.336, -78.413, -1.099]
  MoveL 941 to (-90.26, -236.52, -4.17) mm, rotated rx -180 ry 0 rz 0 deg; joints [6.025, -45.544, 124.902, 6.143, -78.548, -0.86]
  MoveC 942 to (-90.44, -236.97, -4.18) mm, rotated rx -180 ry 0 rz 0 deg; joints [6.004, -45.54, 124.891, 6.121, -78.54, -0.857] to (-90.89, -237.15, -4.17) mm, rotated rx -180 ry 0 rz 0 deg; joints [5.993, -45.528, 124.857, 6.111, -78.518, -0.857]
  MoveL 943 to (-91.53, -237.15, -4.18) mm, rotated rx -180 ry 0 rz 0 deg; joints [5.99, -45.511, 124.806, 6.108, -78.485, -0.86]
  MoveC 944 to (-91.98, -237.15, -3.99) mm, rotated rx -180 ry 0 rz 0 deg; joints [5.988, -45.512, 124.774, 6.107, -78.452, -0.864] to (-92.16, -237.15, -3.54) mm, rotated rx -180 ry 0 rz 0 deg; joints [5.987, -45.538, 124.765, 6.107, -78.417, -0.867]
  Set speed (500.0 mm/s)
  MoveL 945 to (-92.16, -237.15, 5) mm, rotated rx -180 ry 0 rz 0 deg; joints [5.984, -46.126, 124.883, 6.115, -77.949, -0.918]
  MoveL 946 to (-92.16, -235.88, 5) mm, rotated rx 180 ry 0 rz 0 deg; joints [6.042, -46.123, 124.872, 6.174, -77.943, -0.93]
  Set speed (25.4 mm/s)
  MoveL 947 to (-92.16, -235.88, 1.83) mm, rotated rx -180 ry 0 rz 0 deg; joints [6.043, -45.904, 124.829, 6.171, -78.118, -0.911]
  MoveL 948 to (-92.16, -235.88, -7.71) mm, rotated rx -180 ry 0 rz 0 deg; joints [6.046, -45.246, 124.695, 6.163, -78.638, -0.854]
  MoveC 949 to (-91.98, -235.88, -8.16) mm, rotated rx -180 ry 0 rz 0 deg; joints [6.047, -45.22, 124.703, 6.163, -78.672, -0.851] to (-91.53, -235.89, -8.35) mm, rotated rx -180 ry 0 rz 0 deg; joints [6.049, -45.22, 124.736, 6.164, -78.706, -0.847]
  Set speed (50.8 mm/s)
  MoveL 950 to (-90.89, -235.88, -8.35) mm, rotated rx -180 ry 0 rz 0 deg; joints [6.053, -45.237, 124.786, 6.167, -78.739, -0.844]
  MoveC 951 to (-90.44, -236.07, -8.35) mm, rotated rx -180 ry 0 rz 0 deg; joints [6.046, -45.249, 124.823, 6.16, -78.763, -0.84] to (-90.26, -236.52, -8.35) mm, rotated rx 180 ry 0 rz 0 deg; joints [6.026, -45.255, 124.842, 6.139, -78.775, -0.835]
  MoveL 952 to (-90.26, -261.92, -8.35) mm, rotated rx 180 ry 0 rz 0 deg; joints [4.856, -45.309, 125.031, 4.944, -78.889, -0.609]
  MoveL 953 to (-141.06, -261.92, -8.35) mm, rotated rx -180 ry 0 rz 0 deg; joints [4.665, -43.891, 120.959, 4.798, -76.242, -0.8]
  MoveL 954 to (-141.06, -211.12, -8.35) mm, rotated rx 180 ry 0 rz 0 deg; joints [6.91, -43.762, 120.546, 7.117, -76.012, -1.351]
  MoveL 955 to (-90.26, -211.12, -8.35) mm, rotated rx 180 ry 0 rz 0 deg; joints [7.192, -45.188, 124.612, 7.331, -78.639, -1.07]
  MoveL 956 to (-90.26, -236.52, -8.35) mm, rotated rx 180 ry 0 rz 0 deg; joints [6.026, -45.255, 124.842, 6.139, -78.775, -0.835]
  MoveC 957 to (-90.44, -236.97, -8.35) mm, rotated rx -180 ry 0 rz 0 deg; joints [6.005, -45.251, 124.831, 6.118, -78.768, -0.832] to (-90.89, -237.16, -8.35) mm, rotated rx -180 ry 0 rz 0 deg; joints [5.994, -45.24, 124.797, 6.107, -78.745, -0.833]
  MoveL 958 to (-91.53, -237.16, -8.35) mm, rotated rx -180 ry 0 rz 0 deg; joints [5.991, -45.223, 124.746, 6.105, -78.712, -0.836]
  MoveC 959 to (-91.98, -237.16, -8.16) mm, rotated rx 180 ry 0 rz 0 deg; joints [5.989, -45.224, 124.714, 6.103, -78.679, -0.839] to (-92.16, -237.15, -7.72) mm, rotated rx -180 ry 0 rz 0 deg; joints [5.988, -45.25, 124.705, 6.103, -78.645, -0.843]
  Set speed (500.0 mm/s)
  MoveL 960 to (-92.16, -237.16, 6) mm, rotated rx -180 ry 0 rz 0 deg; joints [5.984, -46.195, 124.896, 6.116, -77.894, -0.924]
  MoveL 961 to (-92.16, -54.85, 6) mm, rotated rx -180 ry 0 rz 0 deg; joints [14.171, -45.366, 122.346, 14.575, -76.514, -2.978]
  Set speed (25.4 mm/s)
  MoveL 962 to (-92.16, -54.85, -3.54) mm, rotated rx 180 ry 0 rz 0 deg; joints [14.174, -44.729, 122.217, 14.549, -77.007, -2.848]
  MoveC 963 to (-91.98, -54.85, -3.99) mm, rotated rx -180 ry 0 rz 0 deg; joints [14.177, -44.704, 122.226, 14.549, -77.039, -2.839] to (-91.53, -54.85, -4.17) mm, rotated rx -180 ry 0 rz 0 deg; joints [14.182, -44.704, 122.258, 14.552, -77.071, -2.832]
  Set speed (50.8 mm/s)
  MoveL 964 to (-90.89, -54.85, -4.18) mm, rotated rx -180 ry 0 rz 0 deg; joints [14.189, -44.722, 122.308, 14.558, -77.102, -2.825]
  MoveC 965 to (-90.44, -55.04, -4.18) mm, rotated rx -180 ry 0 rz 0 deg; joints [14.185, -44.736, 122.347, 14.553, -77.126, -2.818] to (-90.26, -55.49, -4.17) mm, rotated rx -180 ry 0 rz 0 deg; joints [14.168, -44.744, 122.371, 14.534, -77.14, -2.811]
  MoveL 966 to (-90.26, -80.89, -4.17) mm, rotated rx -180 ry 0 rz 0 deg; joints [13.052, -44.901, 122.85, 13.375, -77.396, -2.496]
  MoveL 967 to (-141.06, -80.89, -4.17) mm, rotated rx -180 ry 0 rz 0 deg; joints [12.553, -43.433, 118.806, 13.006, -74.862, -2.986]
  MoveL 968 to (-141.06, -30.09, -4.18) mm, rotated rx 180 ry 0 rz 0 deg; joints [14.695, -43.09, 117.82, 15.266, -74.373, -3.705]
  MoveL 969 to (-90.26, -30.09, -4.17) mm, rotated rx 180 ry 0 rz 0 deg; joints [15.272, -44.572, 121.851, 15.687, -76.868, -3.141]
  MoveL 970 to (-90.26, -55.49, -4.17) mm, rotated rx -180 ry 0 rz 0 deg; joints [14.168, -44.744, 122.371, 14.534, -77.14, -2.811]
  MoveC 971 to (-90.44, -55.94, -4.17) mm, rotated rx 180 ry 0 rz 0 deg; joints [14.146, -44.742, 122.365, 14.512, -77.136, -2.807] to (-90.89, -56.12, -4.18) mm, rotated rx -180 ry 0 rz 0 deg; joints [14.133, -44.73, 122.333, 14.5, -77.115, -2.809]
  MoveL 972 to (-91.53, -56.12, -4.17) mm, rotated rx 180 ry 0 rz 0 deg; joints [14.126, -44.712, 122.283, 14.495, -77.084, -2.816]
  MoveC 973 to (-91.98, -56.12, -3.99) mm, rotated rx -180 ry 0 rz 0 deg; joints [14.121, -44.712, 122.251, 14.491, -77.052, -2.823] to (-92.16, -56.12, -3.54) mm, rotated rx -180 ry 0 rz 0 deg; joints [14.119, -44.737, 122.242, 14.491, -77.02, -2.831]
  Set speed (500.0 mm/s)
  MoveL 974 to (-92.16, -56.12, 5) mm, rotated rx 180 ry 0 rz 0 deg; joints [14.116, -45.307, 122.358, 14.515, -76.579, -2.948]
  MoveL 975 to (-92.16, -54.85, 5) mm, rotated rx 180 ry 0 rz 0 deg; joints [14.171, -45.299, 122.333, 14.572, -76.566, -2.964]
  Set speed (25.4 mm/s)
  MoveL 976 to (-92.16, -54.85, 1.82) mm, rotated rx -180 ry 0 rz 0 deg; joints [14.172, -45.087, 122.291, 14.564, -76.731, -2.921]
  MoveL 977 to (-92.16, -54.85, -7.72) mm, rotated rx -180 ry 0 rz 0 deg; joints [14.176, -44.45, 122.159, 14.538, -77.221, -2.791]
  MoveC 978 to (-91.98, -54.85, -8.16) mm, rotated rx -180 ry 0 rz 0 deg; joints [14.178, -44.425, 122.167, 14.538, -77.253, -2.783] to (-91.53, -54.85, -8.35) mm, rotated rx -180 ry 0 rz 0 deg; joints [14.183, -44.425, 122.2, 14.541, -77.285, -2.776]
  Set speed (50.8 mm/s)
  MoveL 979 to (-90.89, -54.85, -8.35) mm, rotated rx -180 ry 0 rz 0 deg; joints [14.19, -44.442, 122.249, 14.547, -77.316, -2.769]
  MoveC 980 to (-90.44, -55.04, -8.35) mm, rotated rx -180 ry 0 rz 0 deg; joints [14.187, -44.456, 122.288, 14.542, -77.34, -2.762] to (-90.26, -55.49, -8.35) mm, rotated rx -180 ry 0 rz 0 deg; joints [14.169, -44.464, 122.312, 14.523, -77.354, -2.754]
  MoveL 981 to (-90.26, -80.89, -8.35) mm, rotated rx -180 ry 0 rz 0 deg; joints [13.054, -44.619, 122.791, 13.365, -77.613, -2.444]
  MoveL 982 to (-141.06, -80.89, -8.35) mm, rotated rx -180 ry 0 rz 0 deg; joints [12.554, -43.165, 118.749, 12.994, -75.068, -2.937]
  MoveL 983 to (-141.06, -30.09, -8.35) mm, rotated rx -180 ry 0 rz 0 deg; joints [14.696, -42.824, 117.762, 15.252, -74.574, -3.648]
  MoveL 984 to (-90.26, -30.09, -8.35) mm, rotated rx 180 ry 0 rz 0 deg; joints [15.274, -44.294, 121.793, 15.675, -77.079, -3.081]
  MoveL 985 to (-90.26, -55.49, -8.35) mm, rotated rx -180 ry 0 rz 0 deg; joints [14.169, -44.464, 122.312, 14.523, -77.354, -2.754]
  MoveC 986 to (-90.44, -55.94, -8.35) mm, rotated rx 180 ry 0 rz 0 deg; joints [14.148, -44.462, 122.306, 14.501, -77.35, -2.75] to (-90.89, -56.12, -8.35) mm, rotated rx -180 ry 0 rz 0 deg; joints [14.135, -44.45, 122.274, 14.489, -77.329, -2.753]
  MoveL 987 to (-91.53, -56.12, -8.35) mm, rotated rx -180 ry 0 rz 0 deg; joints [14.128, -44.433, 122.225, 14.484, -77.298, -2.76]
  MoveC 988 to (-91.98, -56.12, -8.16) mm, rotated rx 180 ry 0 rz 0 deg; joints [14.123, -44.433, 122.192, 14.48, -77.266, -2.767] to (-92.16, -56.12, -7.72) mm, rotated rx -180 ry 0 rz 0 deg; joints [14.12, -44.458, 122.184, 14.48, -77.234, -2.775]
  Set speed (500.0 mm/s)
  MoveL 989 to (-92.16, -56.12, 6) mm, rotated rx -180 ry 0 rz 0 deg; joints [14.115, -45.374, 122.371, 14.517, -76.527, -2.961]
  MoveL 990 to (-219.16, -54.85, 6) mm, rotated rx 180 ry 0 rz 0 deg; joints [12.896, -41.393, 112.003, 13.711, -70.251, -4.241]
  Set speed (25.4 mm/s)
  MoveL 991 to (-219.16, -54.85, -3.54) mm, rotated rx 180 ry 0 rz 0 deg; joints [12.899, -40.824, 111.882, 13.677, -70.686, -4.13]
  MoveC 992 to (-218.98, -54.85, -3.99) mm, rotated rx 180 ry 0 rz 0 deg; joints [12.901, -40.803, 111.892, 13.676, -70.716, -4.123] to (-218.53, -54.85, -4.17) mm, rotated rx 180 ry 0 rz 0 deg; joints [12.905, -40.807, 111.927, 13.678, -70.747, -4.116]
  Set speed (50.8 mm/s)
  MoveL 993 to (-217.89, -54.85, -4.17) mm, rotated rx -180 ry 0 rz 0 deg; joints [12.911, -40.828, 111.981, 13.681, -70.779, -4.11]
  MoveC 994 to (-217.44, -55.04, -4.18) mm, rotated rx -180 ry 0 rz 0 deg; joints [12.907, -40.844, 112.023, 13.676, -70.803, -4.103] to (-217.26, -55.49, -4.17) mm, rotated rx 180 ry 0 rz 0 deg; joints [12.891, -40.854, 112.047, 13.657, -70.817, -4.094]
  MoveL 995 to (-217.26, -80.89, -4.17) mm, rotated rx -180 ry 0 rz 0 deg; joints [11.87, -41.027, 112.515, 12.556, -71.03, -3.686]
  MoveL 996 to (-268.06, -80.89, -4.18) mm, rotated rx -180 ry 0 rz 0 deg; joints [11.454, -39.285, 108.148, 12.323, -68.437, -4.142]
  MoveL 997 to (-268.06, -30.09, -4.18) mm, rotated rx -180 ry 0 rz 0 deg; joints [13.422, -38.91, 107.174, 14.49, -68.02, -5.045]
  MoveL 998 to (-217.26, -30.09, -4.18) mm, rotated rx 180 ry 0 rz 0 deg; joints [13.904, -40.665, 111.539, 14.754, -70.588, -4.515]
  MoveL 999 to (-217.26, -55.49, -4.17) mm, rotated rx 180 ry 0 rz 0 deg; joints [12.891, -40.854, 112.047, 13.657, -70.817, -4.094]
  MoveC 1000 to (-217.44, -55.94, -4.18) mm, rotated rx -180 ry 0 rz 0 deg; joints [12.871, -40.851, 112.04, 13.637, -70.811, -4.088] to (-217.89, -56.12, -4.17) mm, rotated rx -180 ry 0 rz 0 deg; joints [12.86, -40.837, 112.005, 13.626, -70.79, -4.089]
  MoveL 1001 to (-218.53, -56.12, -4.18) mm, rotated rx -180 ry 0 rz 0 deg; joints [12.854, -40.816, 111.952, 13.623, -70.758, -4.096]
  MoveC 1002 to (-218.98, -56.12, -3.99) mm, rotated rx -180 ry 0 rz 0 deg; joints [12.85, -40.812, 111.916, 13.621, -70.727, -4.102] to (-219.16, -56.12, -3.54) mm, rotated rx -180 ry 0 rz 0 deg; joints [12.848, -40.833, 111.906, 13.622, -70.697, -4.109]
  Set speed (500.0 mm/s)
  MoveL 1003 to (-219.16, -56.12, 5) mm, rotated rx -180 ry 0 rz 0 deg; joints [12.845, -41.343, 112.015, 13.652, -70.308, -4.208]
  MoveL 1004 to (-219.16, -54.85, 5) mm, rotated rx 180 ry 0 rz 0 deg; joints [12.896, -41.333, 111.991, 13.707, -70.297, -4.23]
  Set speed (25.4 mm/s)
  MoveL 1005 to (-219.16, -54.85, 1.82) mm, rotated rx -180 ry 0 rz 0 deg; joints [12.897, -41.144, 111.951, 13.696, -70.442, -4.192]
  MoveL 1006 to (-219.16, -54.85, -7.72) mm, rotated rx 180 ry 0 rz 0 deg; joints [12.9, -40.574, 111.827, 13.662, -70.875, -4.082]
  MoveC 1007 to (-218.98, -54.85, -8.16) mm, rotated rx -180 ry 0 rz 0 deg; joints [12.902, -40.553, 111.836, 13.661, -70.905, -4.075] to (-218.53, -54.85, -8.35) mm, rotated rx -180 ry 0 rz 0 deg; joints [12.906, -40.557, 111.872, 13.663, -70.936, -4.068]
  Set speed (50.8 mm/s)
  MoveL 1008 to (-217.89, -54.85, -8.35) mm, rotated rx 180 ry 0 rz 0 deg; joints [12.912, -40.578, 111.925, 13.667, -70.968, -4.062]
  MoveC 1009 to (-217.44, -55.04, -8.35) mm, rotated rx -180 ry 0 rz 0 deg; joints [12.909, -40.594, 111.967, 13.661, -70.993, -4.055] to (-217.26, -55.49, -8.35) mm, rotated rx -180 ry 0 rz 0 deg; joints [12.892, -40.604, 111.991, 13.643, -71.006, -4.045]
  MoveL 1010 to (-217.26, -80.89, -8.35) mm, rotated rx -180 ry 0 rz 0 deg; joints [11.871, -40.775, 112.459, 12.543, -71.221, -3.642]
  MoveL 1011 to (-268.06, -80.89, -8.35) mm, rotated rx 180 ry 0 rz 0 deg; joints [11.455, -39.043, 108.093, 12.309, -68.619, -4.1]
  MoveL 1012 to (-268.06, -30.09, -8.35) mm, rotated rx -180 ry 0 rz 0 deg; joints [13.423, -38.671, 107.119, 14.473, -68.199, -4.996]
  MoveL 1013 to (-217.26, -30.09, -8.35) mm, rotated rx 180 ry 0 rz 0 deg; joints [13.906, -40.416, 111.483, 14.739, -70.776, -4.463]
  MoveL 1014 to (-217.26, -55.49, -8.35) mm, rotated rx -180 ry 0 rz 0 deg; joints [12.892, -40.604, 111.991, 13.643, -71.006, -4.045]
  MoveC 1015 to (-217.44, -55.94, -8.35) mm, rotated rx -180 ry 0 rz 0 deg; joints [12.873, -40.601, 111.984, 13.622, -71.001, -4.04] to (-217.89, -56.12, -8.35) mm, rotated rx -180 ry 0 rz 0 deg; joints [12.861, -40.587, 111.95, 13.612, -70.979, -4.041]
  MoveL 1016 to (-218.53, -56.12, -8.35) mm, rotated rx -180 ry 0 rz 0 deg; joints [12.855, -40.566, 111.896, 13.608, -70.947, -4.048]
  MoveC 1017 to (-218.98, -56.12, -8.16) mm, rotated rx -180 ry 0 rz 0 deg; joints [12.851, -40.562, 111.861, 13.607, -70.916, -4.054] to (-219.16, -56.12, -7.72) mm, rotated rx -180 ry 0 rz 0 deg; joints [12.849, -40.583, 111.851, 13.607, -70.886, -4.061]
  Set speed (500.0 mm/s)
  MoveL 1018 to (-219.16, -56.12, 6) mm, rotated rx -180 ry 0 rz 0 deg; joints [12.845, -41.402, 112.028, 13.656, -70.262, -4.22]
  MoveL 1019 to (-346.16, -54.85, 6) mm, rotated rx 180 ry 0 rz 0 deg; joints [11.828, -36.735, 100.758, 13.206, -63.748, -5.471]
  Set speed (25.4 mm/s)
  MoveL 1020 to (-346.16, -54.85, -3.54) mm, rotated rx -180 ry 0 rz 0 deg; joints [11.831, -36.219, 100.639, 13.164, -64.136, -5.371]
  MoveC 1021 to (-345.98, -54.85, -3.99) mm, rotated rx -180 ry 0 rz 0 deg; joints [11.833, -36.202, 100.651, 13.163, -64.164, -5.365] to (-345.53, -54.85, -4.17) mm, rotated rx -180 ry 0 rz 0 deg; joints [11.836, -36.209, 100.69, 13.163, -64.195, -5.359]
  Set speed (50.8 mm/s)
  MoveL 1022 to (-344.89, -54.85, -4.18) mm, rotated rx -180 ry 0 rz 0 deg; joints [11.841, -36.234, 100.749, 13.165, -64.229, -5.352]
  MoveC 1023 to (-344.44, -55.04, -4.17) mm, rotated rx -180 ry 0 rz 0 deg; joints [11.838, -36.253, 100.794, 13.158, -64.254, -5.344] to (-344.26, -55.49, -4.17) mm, rotated rx -180 ry 0 rz 0 deg; joints [11.822, -36.264, 100.82, 13.14, -64.267, -5.333]
  MoveL 1024 to (-344.26, -80.89, -4.17) mm, rotated rx -180 ry 0 rz 0 deg; joints [10.881, -36.452, 101.29, 12.071, -64.455, -4.829]
  MoveL 1025 to (-395.06, -80.89, -4.17) mm, rotated rx 180 ry 0 rz 0 deg; joints [10.53, -34.405, 96.475, 11.972, -61.714, -5.304]
  MoveL 1026 to (-395.06, -30.09, -4.17) mm, rotated rx -180 ry 0 rz 0 deg; joints [12.349, -33.997, 95.482, 14.1, -61.339, -6.407]
  MoveL 1027 to (-344.26, -30.09, -4.18) mm, rotated rx 180 ry 0 rz 0 deg; joints [12.757, -36.058, 100.309, 14.208, -64.066, -5.849]
  MoveL 1028 to (-344.26, -55.49, -4.17) mm, rotated rx -180 ry 0 rz 0 deg; joints [11.822, -36.264, 100.82, 13.14, -64.267, -5.333]
  MoveC 1029 to (-344.44, -55.94, -4.17) mm, rotated rx 180 ry 0 rz 0 deg; joints [11.804, -36.26, 100.811, 13.121, -64.261, -5.326] to (-344.89, -56.12, -4.17) mm, rotated rx -180 ry 0 rz 0 deg; joints [11.794, -36.244, 100.773, 13.112, -64.238, -5.327]
  MoveL 1030 to (-345.53, -56.12, -4.18) mm, rotated rx -180 ry 0 rz 0 deg; joints [11.789, -36.219, 100.714, 13.11, -64.205, -5.333]
  MoveC 1031 to (-345.98, -56.12, -3.99) mm, rotated rx -180 ry 0 rz 0 deg; joints [11.786, -36.212, 100.675, 13.109, -64.173, -5.339] to (-346.16, -56.12, -3.54) mm, rotated rx 180 ry 0 rz 0 deg; joints [11.784, -36.229, 100.664, 13.111, -64.145, -5.346]
  Set speed (500.0 mm/s)
  MoveL 1032 to (-346.16, -56.12, 5) mm, rotated rx -180 ry 0 rz 0 deg; joints [11.782, -36.691, 100.77, 13.148, -63.799, -5.435]
  MoveL 1033 to (-346.16, -54.85, 5) mm, rotated rx -180 ry 0 rz 0 deg; joints [11.828, -36.681, 100.746, 13.201, -63.789, -5.461]
  Set speed (25.4 mm/s)
  MoveL 1034 to (-346.16, -54.85, 1.82) mm, rotated rx -180 ry 0 rz 0 deg; joints [11.829, -36.51, 100.707, 13.187, -63.918, -5.427]
  MoveL 1035 to (-346.16, -54.85, -7.71) mm, rotated rx 180 ry 0 rz 0 deg; joints [11.832, -35.992, 100.585, 13.147, -64.304, -5.328]
  MoveC 1036 to (-345.98, -54.85, -8.16) mm, rotated rx -180 ry 0 rz 0 deg; joints [11.834, -35.975, 100.596, 13.145, -64.332, -5.322] to (-345.53, -54.85, -8.35) mm, rotated rx 180 ry 0 rz 0 deg; joints [11.837, -35.982, 100.635, 13.146, -64.363, -5.316]
  Set speed (50.8 mm/s)
  MoveL 1037 to (-344.89, -54.85, -8.35) mm, rotated rx -180 ry 0 rz 0 deg; joints [11.842, -36.007, 100.694, 13.147, -64.397, -5.309]
  MoveC 1038 to (-344.44, -55.04, -8.35) mm, rotated rx -180 ry 0 rz 0 deg; joints [11.839, -36.026, 100.74, 13.141, -64.422, -5.301] to (-344.26, -55.49, -8.35) mm, rotated rx -180 ry 0 rz 0 deg; joints [11.824, -36.037, 100.766, 13.122, -64.435, -5.29]
  MoveL 1039 to (-344.26, -80.89, -8.35) mm, rotated rx -180 ry 0 rz 0 deg; joints [10.882, -36.224, 101.236, 12.055, -64.624, -4.79]
  MoveL 1040 to (-395.06, -80.89, -8.35) mm, rotated rx -180 ry 0 rz 0 deg; joints [10.531, -34.185, 96.42, 11.954, -61.876, -5.266]
  MoveL 1041 to (-395.06, -30.09, -8.35) mm, rotated rx 180 ry 0 rz 0 deg; joints [12.35, -33.778, 95.427, 14.08, -61.498, -6.362]
  MoveL 1042 to (-344.26, -30.09, -8.35) mm, rotated rx 180 ry 0 rz 0 deg; joints [12.758, -35.832, 100.255, 14.189, -64.233, -5.803]
  MoveL 1043 to (-344.26, -55.49, -8.35) mm, rotated rx -180 ry 0 rz 0 deg; joints [11.824, -36.037, 100.766, 13.122, -64.435, -5.29]
  MoveC 1044 to (-344.44, -55.94, -8.35) mm, rotated rx 180 ry 0 rz 0 deg; joints [11.806, -36.033, 100.757, 13.103, -64.429, -5.283] to (-344.89, -56.12, -8.35) mm, rotated rx -180 ry 0 rz 0 deg; joints [11.795, -36.017, 100.719, 13.094, -64.407, -5.284]
  MoveL 1045 to (-345.53, -56.12, -8.35) mm, rotated rx -180 ry 0 rz 0 deg; joints [11.79, -35.992, 100.66, 13.092, -64.373, -5.29]
  MoveC 1046 to (-345.98, -56.12, -8.16) mm, rotated rx 180 ry 0 rz 0 deg; joints [11.787, -35.985, 100.621, 13.092, -64.341, -5.297] to (-346.16, -56.12, -7.72) mm, rotated rx 180 ry 0 rz 0 deg; joints [11.785, -36.002, 100.609, 13.093, -64.313, -5.303]
  Set speed (500.0 mm/s)
  MoveL 1047 to (-346.16, -56.12, 15) mm, rotated rx -180 ry 0 rz 0 deg; joints [11.779, -37.23, 100.888, 13.192, -63.388, -5.54]
  Print: /'2D Contour1'
  Set speed (500.0 mm/s)
  MoveL 1048 to (-12.15, 15.92, 15) mm, rotated rx 180 ry 0 rz 0 deg; joints [18.325, -47.664, 127.03, 18.672, -79.043, -3.115]
  MoveL 1049 to (-12.15, 15.92, 6) mm, rotated rx -180 ry 0 rz 0 deg; joints [18.329, -47.029, 126.913, 18.644, -79.533, -2.947]
  Set speed (25.4 mm/s)
  MoveL 1050 to (-12.15, 15.92, -4.37) mm, rotated rx -180 ry 0 rz 0 deg; joints [18.334, -46.296, 126.768, 18.615, -80.091, -2.757]
  MoveC 1051 to (-12.34, 15.92, -4.81) mm, rotated rx 180 ry 0 rz 0 deg; joints [18.331, -46.26, 126.748, 18.612, -80.106, -2.751] to (-12.79, 15.92, -5) mm, rotated rx 180 ry 0 rz 0 deg; joints [18.325, -46.235, 126.711, 18.606, -80.094, -2.754]
  Set speed (50.8 mm/s)
  MoveL 1052 to (-13.42, 15.92, -5) mm, rotated rx 180 ry 0 rz 0 deg; joints [18.315, -46.22, 126.664, 18.598, -80.064, -2.763]
  MoveC 1053 to (-13.87, 16.1, -5) mm, rotated rx -180 ry 0 rz 0 deg; joints [18.317, -46.207, 126.626, 18.601, -80.04, -2.771] to (-14.06, 16.55, -5) mm, rotated rx -180 ry 0 rz 0 deg; joints [18.334, -46.199, 126.601, 18.62, -80.025, -2.78]
  MoveL 1054 to (-14.06, 168.95, -5) mm, rotated rx 180 ry 0 rz 0 deg; joints [24.853, -44.75, 122.138, 25.47, -77.706, -5.116]
  MoveL 1055 to (-39.46, 168.95, -5) mm, rotated rx 180 ry 0 rz 0 deg; joints [24.382, -44.066, 120.257, 25.106, -76.578, -5.541]
  MoveC 1056 to (-52.16, 156.25, -5) mm, rotated rx -180 ry 0 rz 0 deg; joints [23.643, -43.862, 119.726, 24.383, -76.207, -5.515] to (-64.86, 168.95, -5) mm, rotated rx 180 ry 0 rz 0 deg; joints [23.927, -43.356, 118.345, 24.766, -75.44, -5.957]
  MoveL 1057 to (-90.26, 168.95, -5) mm, rotated rx 180 ry 0 rz 0 deg; joints [23.488, -42.621, 116.403, 24.45, -74.294, -6.367]
  MoveL 1058 to (-166.46, 168.95, -5) mm, rotated rx 180 ry 0 rz 0 deg; joints [22.257, -40.261, 110.374, 23.64, -70.788, -7.568]
  MoveC 1059 to (-179.16, 156.25, -5) mm, rotated rx -180 ry 0 rz 0 deg; joints [21.59, -40.004, 109.753, 22.99, -70.363, -7.498] to (-191.86, 168.95, -5) mm, rotated rx -180 ry 0 rz 0 deg; joints [21.874, -39.421, 108.292, 23.415, -69.595, -7.965]
  MoveL 1060 to (-293.46, 168.95, -5) mm, rotated rx 180 ry 0 rz 0 deg; joints [20.459, -35.781, 99.538, 22.743, -64.668, -9.572]
  MoveC 1061 to (-306.16, 156.25, -5) mm, rotated rx -180 ry 0 rz 0 deg; joints [19.851, -35.465, 98.81, 22.154, -64.184, -9.469] to (-318.86, 168.95, -5) mm, rotated rx 180 ry 0 rz 0 deg; joints [20.132, -34.795, 97.229, 22.634, -63.39, -9.988]
  MoveL 1062 to (-395.06, 168.95, -5) mm, rotated rx 180 ry 0 rz 0 deg; joints [19.209, -31.628, 89.949, 22.462, -59.416, -11.304]
  MoveL 1063 to (-420.46, 168.95, -5) mm, rotated rx -180 ry 0 rz 0 deg; joints [18.919, -30.496, 87.386, 22.461, -58.036, -11.775]
  MoveC 1064 to (-433.16, 156.25, -5) mm, rotated rx -180 ry 0 rz 0 deg; joints [18.363, -30.104, 86.517, 21.931, -57.478, -11.653] to (-445.86, 168.95, -5) mm, rotated rx -180 ry 0 rz 0 deg; joints [18.638, -29.319, 84.745, 22.494, -56.623, -12.268]
  MoveL 1065 to (-471.26, 168.95, -5) mm, rotated rx -180 ry 0 rz 0 deg; joints [18.364, -28.094, 82.017, 22.562, -55.173, -12.787]
  MoveL 1066 to (-471.26, 16.55, -5) mm, rotated rx -180 ry 0 rz 0 deg; joints [13.36, -30.115, 86.667, 16.041, -56.71, -8.489]
  MoveL 1067 to (-14.06, 16.55, -5) mm, rotated rx -180 ry 0 rz 0 deg; joints [18.334, -46.199, 126.601, 18.62, -80.025, -2.78]
  MoveC 1068 to (-13.61, 16.36, -5) mm, rotated rx -180 ry 0 rz 0 deg; joints [18.333, -46.211, 126.639, 18.616, -80.049, -2.771] to (-13.42, 15.92, -5) mm, rotated rx 180 ry 0 rz 0 deg; joints [18.315, -46.22, 126.664, 18.598, -80.064, -2.763]
  MoveL 1069 to (-13.42, 15.28, -5) mm, rotated rx -180 ry 0 rz 0 deg; joints [18.287, -46.224, 126.679, 18.569, -80.073, -2.755]
  MoveC 1070 to (-13.42, 14.83, -4.81) mm, rotated rx -180 ry 0 rz 0 deg; joints [18.267, -46.241, 126.693, 18.548, -80.069, -2.753] to (-13.42, 14.65, -4.37) mm, rotated rx -180 ry 0 rz 0 deg; joints [18.258, -46.274, 126.704, 18.541, -80.048, -2.758]
  Set speed (500.0 mm/s)
  MoveL 1071 to (-13.42, 14.65, 5) mm, rotated rx 180 ry 0 rz 0 deg; joints [18.254, -46.936, 126.835, 18.567, -79.544, -2.929]
  MoveL 1072 to (-12.15, 15.92, 5) mm, rotated rx -180 ry 0 rz 0 deg; joints [18.33, -46.958, 126.899, 18.641, -79.587, -2.929]
  Set speed (25.4 mm/s)
  MoveL 1073 to (-12.15, 15.92, 1) mm, rotated rx 180 ry 0 rz 0 deg; joints [18.332, -46.676, 126.844, 18.63, -79.803, -2.855]
  MoveL 1074 to (-12.15, 15.92, -7.72) mm, rotated rx -180 ry 0 rz 0 deg; joints [18.335, -46.059, 126.719, 18.606, -80.27, -2.696]
  MoveC 1075 to (-12.34, 15.92, -8.16) mm, rotated rx -180 ry 0 rz 0 deg; joints [18.333, -46.023, 126.699, 18.603, -80.285, -2.691] to (-12.79, 15.92, -8.35) mm, rotated rx -180 ry 0 rz 0 deg; joints [18.326, -45.998, 126.662, 18.597, -80.273, -2.693]
  Set speed (50.8 mm/s)
  MoveL 1076 to (-13.42, 15.92, -8.35) mm, rotated rx 180 ry 0 rz 0 deg; joints [18.317, -45.983, 126.615, 18.589, -80.242, -2.702]
  MoveC 1077 to (-13.87, 16.1, -8.35) mm, rotated rx -180 ry 0 rz 0 deg; joints [18.318, -45.97, 126.577, 18.592, -80.218, -2.711] to (-14.06, 16.55, -8.35) mm, rotated rx -180 ry 0 rz 0 deg; joints [18.336, -45.962, 126.552, 18.611, -80.203, -2.719]
  MoveL 1078 to (-14.06, 168.95, -8.35) mm, rotated rx 180 ry 0 rz 0 deg; joints [24.855, -44.526, 122.091, 25.455, -77.866, -5.039]
  MoveL 1079 to (-39.46, 168.95, -8.35) mm, rotated rx -180 ry 0 rz 0 deg; joints [24.383, -43.847, 120.21, 25.09, -76.734, -5.466]
  MoveC 1080 to (-52.16, 156.25, -8.35) mm, rotated rx 180 ry 0 rz 0 deg; joints [23.645, -43.644, 119.68, 24.367, -76.363, -5.442] to (-64.86, 168.95, -8.35) mm, rotated rx -180 ry 0 rz 0 deg; joints [23.929, -43.142, 118.299, 24.749, -75.594, -5.885]
  MoveL 1081 to (-90.26, 168.95, -8.35) mm, rotated rx -180 ry 0 rz 0 deg; joints [23.489, -42.411, 116.357, 24.432, -74.444, -6.296]
  MoveL 1082 to (-166.46, 168.95, -8.35) mm, rotated rx -180 ry 0 rz 0 deg; joints [22.259, -40.063, 110.33, 23.62, -70.929, -7.504]
  MoveC 1083 to (-179.16, 156.25, -8.35) mm, rotated rx -180 ry 0 rz 0 deg; joints [21.591, -39.808, 109.708, 22.97, -70.503, -7.436] to (-191.86, 168.95, -8.35) mm, rotated rx 180 ry 0 rz 0 deg; joints [21.875, -39.227, 108.247, 23.395, -69.733, -7.902]
  MoveL 1084 to (-293.46, 168.95, -8.35) mm, rotated rx -180 ry 0 rz 0 deg; joints [20.46, -35.6, 99.494, 22.72, -64.794, -9.514]
  MoveC 1085 to (-306.16, 156.25, -8.35) mm, rotated rx 180 ry 0 rz 0 deg; joints [19.852, -35.285, 98.766, 22.131, -64.31, -9.412] to (-318.86, 168.95, -8.35) mm, rotated rx -180 ry 0 rz 0 deg; joints [20.133, -34.617, 97.185, 22.61, -63.514, -9.931]
  MoveL 1086 to (-395.06, 168.95, -8.35) mm, rotated rx -180 ry 0 rz 0 deg; joints [19.21, -31.459, 89.904, 22.435, -59.532, -11.249]
  MoveL 1087 to (-420.46, 168.95, -8.35) mm, rotated rx -180 ry 0 rz 0 deg; joints [18.92, -30.328, 87.342, 22.434, -58.149, -11.721]
  MoveC 1088 to (-433.16, 156.25, -8.35) mm, rotated rx 180 ry 0 rz 0 deg; joints [18.364, -29.938, 86.472, 21.904, -57.591, -11.6] to (-445.86, 168.95, -8.35) mm, rotated rx 180 ry 0 rz 0 deg; joints [18.639, -29.154, 84.7, 22.465, -56.733, -12.214]
  MoveL 1089 to (-471.26, 168.95, -8.35) mm, rotated rx -180 ry 0 rz 0 deg; joints [18.365, -27.931, 81.971, 22.532, -55.281, -12.734]
  MoveL 1090 to (-471.26, 16.55, -8.35) mm, rotated rx -180 ry 0 rz 0 deg; joints [13.361, -29.948, 86.622, 16.02, -56.827, -8.45]
  MoveL 1091 to (-14.06, 16.55, -8.35) mm, rotated rx 180 ry 0 rz 0 deg; joints [18.336, -45.962, 126.552, 18.611, -80.203, -2.719]
  MoveC 1092 to (-13.61, 16.36, -8.35) mm, rotated rx -180 ry 0 rz 0 deg; joints [18.334, -45.975, 126.59, 18.608, -80.227, -2.71] to (-13.42, 15.92, -8.35) mm, rotated rx 180 ry 0 rz 0 deg; joints [18.317, -45.983, 126.615, 18.589, -80.242, -2.702]
  MoveL 1093 to (-13.42, 15.28, -8.35) mm, rotated rx -180 ry 0 rz 0 deg; joints [18.288, -45.987, 126.63, 18.56, -80.251, -2.694]
  MoveC 1094 to (-13.42, 14.83, -8.16) mm, rotated rx -180 ry 0 rz 0 deg; joints [18.268, -46.004, 126.644, 18.539, -80.247, -2.692] to (-13.42, 14.65, -7.72) mm, rotated rx -180 ry 0 rz 0 deg; joints [18.26, -46.037, 126.655, 18.532, -80.226, -2.698]
  Set speed (500.0 mm/s)
  MoveL 1095 to (-13.42, 14.65, 6) mm, rotated rx 180 ry 0 rz 0 deg; joints [18.254, -47.006, 126.849, 18.57, -79.49, -2.948]
  MoveL 1096 to (18.41, 14.65, 6) mm, rotated rx 180 ry 0 rz 0 deg; joints [18.735, -47.807, 129.213, 18.971, -80.997, -2.512]
  Set speed (25.4 mm/s)
  MoveL 1097 to (18.41, 14.65, -4.37) mm, rotated rx -180 ry 0 rz 0 deg; joints [18.74, -47.051, 129.066, 18.946, -81.572, -2.313]
  MoveC 1098 to (18.41, 14.83, -4.81) mm, rotated rx -180 ry 0 rz 0 deg; joints [18.748, -47.017, 129.054, 18.953, -81.594, -2.307] to (18.41, 15.28, -5) mm, rotated rx -180 ry 0 rz 0 deg; joints [18.769, -47, 129.041, 18.974, -81.598, -2.308]
  Set speed (50.8 mm/s)
  MoveL 1099 to (18.41, 15.92, -5) mm, rotated rx -180 ry 0 rz 0 deg; joints [18.798, -46.995, 129.025, 19.004, -81.588, -2.316]
  MoveC 1100 to (18.6, 16.36, -5) mm, rotated rx -180 ry 0 rz 0 deg; joints [18.821, -46.996, 129.027, 19.027, -81.591, -2.319] to (19.04, 16.55, -5) mm, rotated rx 180 ry 0 rz 0 deg; joints [18.837, -47.006, 129.056, 19.042, -81.61, -2.314]
  MoveL 1101 to (39.46, 16.55, -5) mm, rotated rx -180 ry 0 rz 0 deg; joints [19.16, -47.478, 130.549, 19.322, -82.587, -2.016]
  MoveL 1102 to (471.26, 16.55, -5) mm, rotated rx 180 ry 0 rz 30 deg; joints [37.537, -51.906, 150.133, 67.627, -92.253, 7.406]
  MoveL 1103 to (471.26, 168.95, -5) mm, rotated rx 180 ry 0 rz 0 deg; joints [38.595, -52.001, 153.051, 39.008, -97.753, 7.202]
  MoveL 1104 to (445.86, 168.95, -5) mm, rotated rx 180 ry 0 rz 0 deg; joints [37.562, -51.972, 151.669, 37.866, -96.809, 6.208]
  MoveC 1105 to (433.16, 156.25, -5) mm, rotated rx 180 ry 0 rz 0 deg; joints [36.403, -51.942, 151.491, 36.695, -96.808, 5.962] to (420.46, 168.95, -5) mm, rotated rx -180 ry 0 rz 0 deg; joints [36.575, -51.893, 150.259, 36.788, -95.845, 5.272]
  MoveL 1106 to (395.06, 168.95, -5) mm, rotated rx -180 ry 0 rz 0 deg; joints [35.631, -51.767, 148.821, 35.771, -94.862, 4.39]
  MoveL 1107 to (318.86, 168.95, -5) mm, rotated rx 180 ry 0 rz 0 deg; joints [33.041, -51.128, 144.348, 33.052, -91.83, 2.028]
  MoveC 1108 to (306.16, 156.25, -5) mm, rotated rx 180 ry 0 rz 0 deg; joints [32.02, -51.06, 144.065, 32.028, -91.678, 1.866] to (293.46, 168.95, -5) mm, rotated rx -180 ry 0 rz 0 deg; joints [32.251, -50.835, 142.805, 32.246, -90.797, 1.323]
  MoveL 1109 to (191.86, 168.95, -5) mm, rotated rx -180 ry 0 rz 0 deg; joints [29.403, -49.311, 136.386, 29.452, -86.583, -1.166]
  MoveC 1110 to (179.16, 156.25, -5) mm, rotated rx 180 ry 0 rz 0 deg; joints [28.498, -49.197, 136.012, 28.554, -86.332, -1.25] to (166.46, 168.95, -5) mm, rotated rx -180 ry 0 rz 0 deg; joints [28.761, -48.849, 134.719, 28.85, -85.511, -1.719]
  MoveL 1111 to (90.26, 168.95, -5) mm, rotated rx -180 ry 0 rz 0 deg; joints [26.981, -47.287, 129.57, 27.242, -82.259, -3.252]
  MoveL 1112 to (64.86, 168.95, -5) mm, rotated rx -180 ry 0 rz 0 deg; joints [26.433, -46.711, 127.802, 26.768, -81.162, -3.727]
  MoveC 1113 to (61.14, 159.97, -5) mm, rotated rx -180 ry 0 rz 0 deg; joints [25.97, -46.719, 127.85, 26.299, -81.165, -3.645] to (52.16, 156.25, -5) mm, rotated rx 180 ry 0 rz 0 deg; joints [25.626, -46.547, 127.342, 25.974, -80.839, -3.746]
  MoveL 1114 to (52.16, 156.25, -5) mm, rotated rx 180 ry 0 rz 0 deg; joints [25.626, -46.547, 127.342, 25.974, -80.839, -3.746]
  MoveC 1115 to (43.18, 159.97, -5) mm, rotated rx 180 ry 0 rz 0 deg; joints [25.601, -46.294, 126.579, 25.986, -80.379, -3.968] to (39.46, 168.95, -5) mm, rotated rx -180 ry 0 rz 0 deg; joints [25.904, -46.107, 126.008, 26.322, -80.057, -4.188]
  MoveL 1116 to (14.06, 168.95, -5) mm, rotated rx -180 ry 0 rz 0 deg; joints [25.395, -45.478, 124.186, 25.903, -78.946, -4.635]
  MoveL 1117 to (14.06, 16.55, -5) mm, rotated rx -180 ry 0 rz 0 deg; joints [18.759, -46.887, 128.688, 18.976, -81.371, -2.386]
  MoveL 1118 to (19.04, 16.55, -5) mm, rotated rx 180 ry 0 rz 0 deg; joints [18.837, -47.006, 129.056, 19.042, -81.61, -2.314]
  MoveC 1119 to (19.49, 16.36, -5) mm, rotated rx -180 ry 0 rz 0 deg; joints [18.835, -47.017, 129.093, 19.039, -81.634, -2.306] to (19.68, 15.92, -5) mm, rotated rx -180 ry 0 rz 0 deg; joints [18.818, -47.025, 129.118, 19.021, -81.649, -2.298]
  MoveL 1120 to (19.68, 15.28, -5) mm, rotated rx -180 ry 0 rz 0 deg; joints [18.789, -47.03, 129.134, 18.991, -81.659, -2.29]
  MoveC 1121 to (19.68, 14.83, -4.81) mm, rotated rx 180 ry 0 rz 0 deg; joints [18.768, -47.047, 129.148, 18.97, -81.655, -2.288] to (19.68, 14.65, -4.37) mm, rotated rx 180 ry 0 rz 0 deg; joints [18.759, -47.081, 129.159, 18.962, -81.633, -2.295]
  Set speed (500.0 mm/s)
  MoveL 1122 to (19.68, 14.65, 5) mm, rotated rx -180 ry 0 rz 0 deg; joints [18.755, -47.765, 129.293, 18.985, -81.113, -2.475]
  MoveL 1123 to (18.41, 14.65, 5) mm, rotated rx -180 ry 0 rz 0 deg; joints [18.735, -47.734, 129.2, 18.969, -81.052, -2.493]
  Set speed (25.4 mm/s)
  MoveL 1124 to (18.41, 14.65, 1) mm, rotated rx 180 ry 0 rz 0 deg; joints [18.737, -47.442, 129.143, 18.958, -81.275, -2.416]
  MoveL 1125 to (18.41, 14.65, -7.72) mm, rotated rx -180 ry 0 rz 0 deg; joints [18.741, -46.806, 129.016, 18.938, -81.756, -2.249]
  MoveC 1126 to (18.41, 14.83, -8.16) mm, rotated rx -180 ry 0 rz 0 deg; joints [18.75, -46.772, 129.005, 18.946, -81.778, -2.243] to (18.41, 15.28, -8.35) mm, rotated rx 180 ry 0 rz 0 deg; joints [18.771, -46.755, 128.991, 18.966, -81.782, -2.245]
  Set speed (50.8 mm/s)
  MoveL 1127 to (18.41, 15.92, -8.35) mm, rotated rx 180 ry 0 rz 0 deg; joints [18.8, -46.751, 128.975, 18.996, -81.773, -2.252]
  MoveC 1128 to (18.6, 16.36, -8.35) mm, rotated rx 180 ry 0 rz 0 deg; joints [18.823, -46.752, 128.977, 19.02, -81.775, -2.255] to (19.04, 16.55, -8.35) mm, rotated rx 180 ry 0 rz 0 deg; joints [18.838, -46.761, 129.006, 19.034, -81.794, -2.25]
  MoveL 1129 to (39.46, 16.55, -8.35) mm, rotated rx -180 ry 0 rz 0 deg; joints [19.162, -47.228, 130.498, 19.315, -82.775, -1.949]
  MoveL 1130 to (471.26, 16.55, -8.35) mm, rotated rx 180 ry 0 rz 30 deg; joints [37.539, -51.554, 150.066, 67.64, -92.361, 7.669]
  MoveL 1131 to (471.26, 168.95, -8.35) mm, rotated rx 180 ry 0 rz 0 deg; joints [38.598, -51.626, 152.979, 39.038, -97.988, 7.395]
  MoveL 1132 to (445.86, 168.95, -8.35) mm, rotated rx -180 ry 0 rz 0 deg; joints [37.564, -51.608, 151.6, 37.891, -97.041, 6.39]
  MoveC 1133 to (433.16, 156.25, -8.35) mm, rotated rx -180 ry 0 rz 0 deg; joints [36.406, -51.58, 151.422, 36.719, -97.042, 6.139] to (420.46, 168.95, -8.35) mm, rotated rx -180 ry 0 rz 0 deg; joints [36.577, -51.54, 150.192, 36.808, -96.072, 5.444]
  MoveL 1134 to (395.06, 168.95, -8.35) mm, rotated rx 180 ry 0 rz 0 deg; joints [35.634, -51.425, 148.755, 35.788, -95.086, 4.552]
  MoveL 1135 to (318.86, 168.95, -8.35) mm, rotated rx 180 ry 0 rz 0 deg; joints [33.044, -50.815, 144.287, 33.059, -92.041, 2.166]
  MoveC 1136 to (306.16, 156.25, -8.35) mm, rotated rx -180 ry 0 rz 0 deg; joints [32.023, -50.749, 144.005, 32.034, -91.891, 1.999] to (293.46, 168.95, -8.35) mm, rotated rx 180 ry 0 rz 0 deg; joints [32.253, -50.531, 142.746, 32.25, -91.004, 1.454]
  MoveL 1137 to (191.86, 168.95, -8.35) mm, rotated rx 180 ry 0 rz 0 deg; joints [29.405, -49.038, 136.332, 29.448, -86.773, -1.058]
  MoveC 1138 to (179.16, 156.25, -8.35) mm, rotated rx -180 ry 0 rz 0 deg; joints [28.5, -48.926, 135.958, 28.55, -86.523, -1.146] to (166.46, 168.95, -8.35) mm, rotated rx 180 ry 0 rz 0 deg; joints [28.763, -48.583, 134.667, 28.844, -85.698, -1.616]
  MoveL 1139 to (90.26, 168.95, -8.35) mm, rotated rx -180 ry 0 rz 0 deg; joints [26.983, -47.041, 129.52, 27.232, -82.434, -3.162]
  MoveL 1140 to (64.86, 168.95, -8.35) mm, rotated rx -180 ry 0 rz 0 deg; joints [26.434, -46.47, 127.753, 26.756, -81.332, -3.641]
  MoveC 1141 to (61.14, 159.97, -8.35) mm, rotated rx -180 ry 0 rz 0 deg; joints [25.972, -46.478, 127.8, 26.287, -81.336, -3.56] to (52.16, 156.25, -8.35) mm, rotated rx -180 ry 0 rz 0 deg; joints [25.627, -46.308, 127.293, 25.962, -81.01, -3.662]
  MoveL 1142 to (52.16, 156.25, -8.35) mm, rotated rx -180 ry 0 rz 0 deg; joints [25.627, -46.308, 127.293, 25.962, -81.01, -3.662]
  MoveC 1143 to (43.18, 159.97, -8.35) mm, rotated rx 180 ry 0 rz 0 deg; joints [25.603, -46.057, 126.53, 25.974, -80.548, -3.885] to (39.46, 168.95, -8.35) mm, rotated rx -180 ry 0 rz 0 deg; joints [25.906, -45.872, 125.959, 26.309, -80.224, -4.104]
  MoveL 1144 to (14.06, 168.95, -8.35) mm, rotated rx 180 ry 0 rz 0 deg; joints [25.397, -45.248, 124.139, 25.889, -79.109, -4.554]
  MoveL 1145 to (14.06, 16.55, -8.35) mm, rotated rx 180 ry 0 rz 0 deg; joints [18.761, -46.644, 128.638, 18.968, -81.554, -2.322]
  MoveL 1146 to (19.04, 16.55, -8.35) mm, rotated rx 180 ry 0 rz 0 deg; joints [18.838, -46.761, 129.006, 19.034, -81.794, -2.25]
  MoveC 1147 to (19.49, 16.36, -8.35) mm, rotated rx -180 ry 0 rz 0 deg; joints [18.837, -46.773, 129.043, 19.032, -81.818, -2.242] to (19.68, 15.92, -8.35) mm, rotated rx -180 ry 0 rz 0 deg; joints [18.819, -46.78, 129.068, 19.013, -81.834, -2.234]
  MoveL 1148 to (19.68, 15.28, -8.35) mm, rotated rx 180 ry 0 rz 0 deg; joints [18.79, -46.785, 129.084, 18.983, -81.843, -2.226]
  MoveC 1149 to (19.68, 14.83, -8.16) mm, rotated rx -180 ry 0 rz 0 deg; joints [18.77, -46.802, 129.098, 18.962, -81.839, -2.225] to (19.68, 14.65, -7.72) mm, rotated rx -180 ry 0 rz 0 deg; joints [18.761, -46.836, 129.109, 18.955, -81.817, -2.231]
  Set speed (500.0 mm/s)
  MoveL 1150 to (19.68, 14.65, 6) mm, rotated rx 180 ry 0 rz 0 deg; joints [18.755, -47.838, 129.307, 18.988, -81.057, -2.494]
  MoveL 1151 to (12.15, -16.75, 6) mm, rotated rx -180 ry 0 rz 0 deg; joints [17.197, -47.88, 129.499, 17.406, -81.127, -2.227]
  Set speed (25.4 mm/s)
  MoveL 1152 to (12.15, -16.75, -4.37) mm, rotated rx -180 ry 0 rz 0 deg; joints [17.202, -47.121, 129.351, 17.383, -81.71, -2.043]
  MoveC 1153 to (12.34, -16.75, -4.81) mm, rotated rx -180 ry 0 rz 0 deg; joints [17.205, -47.093, 129.358, 17.384, -81.744, -2.033] to (12.79, -16.75, -5) mm, rotated rx -180 ry 0 rz 0 deg; joints [17.211, -47.09, 129.389, 17.39, -81.776, -2.023]
  Set speed (50.8 mm/s)
  MoveL 1154 to (13.42, -16.75, -5) mm, rotated rx -180 ry 0 rz 0 deg; joints [17.22, -47.105, 129.436, 17.397, -81.807, -2.015]
  MoveC 1155 to (13.87, -16.94, -5) mm, rotated rx -180 ry 0 rz 0 deg; joints [17.218, -47.117, 129.473, 17.394, -81.832, -2.007] to (14.06, -17.39, -5) mm, rotated rx -180 ry 0 rz 0 deg; joints [17.2, -47.124, 129.497, 17.375, -81.847, -1.999]
  MoveL 1156 to (14.06, -169.79, -5) mm, rotated rx -180 ry 0 rz 0 deg; joints [9.896, -47.875, 132.228, 9.954, -83.567, -0.702]
  MoveL 1157 to (471.26, -169.79, -5) mm, rotated rx 180 ry 0 rz 30 deg; joints [26.904, -51.446, 156.915, 57.661, -97.508, 12.826]
  MoveL 1158 to (471.26, -17.39, -5) mm, rotated rx -180 ry 0 rz 30 deg; joints [35.785, -51.93, 151.533, 65.949, -93.044, 8.564]
  MoveL 1159 to (445.86, -17.39, -5) mm, rotated rx 180 ry 0 rz 30 deg; joints [34.84, -51.847, 150.09, 64.952, -92.613, 7.265]
